// TwinCAT 3 PLC project PLC
// ProgramVersion: 3.1.4023.0
// libraries:
//   Tc2_Standard, * (Beckhoff Automation GmbH)
//   Tc2_System, * (Beckhoff Automation GmbH)
//   Tc3_Module, * (Beckhoff Automation GmbH)
// project tree:
//   / PlcTask.TcTTO
//   POUs/ MAIN.TcPOU
//   DUTs/IO/PdoEntries/ Status_543010BE.TcDUT, Samples_F24E104A.TcDUT, StartTimeNextLatch_02E0C1C8.TcDUT, Status_06143A9F.TcDUT, Status_BA3D1C5D.TcDUT, Status_F2CE6D91.TcDUT, Control_EBEDCF76.TcDUT
//   DUTs/IO/PDOs/ InfoData_6F19DB2B.TcDUT, PAI_Status_Channel_AE4AC104.TcDUT, PAI_Samples_1_Channel_EEA51725.TcDUT, PAI_Timestamp_Channel_6DC4D296.TcDUT, WcState_9091E0EB.TcDUT, InfoData_BEF6B88E.TcDUT, MMS_Device_Inputs_7D6F8734.TcDUT, MMS_Acceleration_Status_11769099.TcDUT, MMS_Acceleration_X_Axis_80E77D6A.TcDUT, MMS_Acceleration_Y_Axis_80E77D6A.TcDUT, MMS_Acceleration_Z_Axis_80E77D6A.TcDUT, MMS_Acceleration_Timestamp_8B9FE1A2.TcDUT, MMS_Voltage_Us_In_Inputs_60D55C72.TcDUT, MMS_Voltage_Up_In_Inputs_60D55C72.TcDUT, MMS_Voltage_Up_Out_Inputs_60D55C72.TcDUT, MMS_Device_Outputs_E6E6F9D1.TcDUT, InfoData_E68C61CD.TcDUT, WcState_0B2B16F9.TcDUT, InfoData_2A97D6CF.TcDUT, Inputs_25A0042B.TcDUT, Outputs_2397A10E.TcDUT
//   DUTs/IO/Boxes/ EK1100_1FC0878B.TcDUT, EK1122_1FC0878B.TcDUT, ELM3002_B416BFEF.TcDUT, ELM3004_9E251EA4.TcDUT, ELM3102_B416BFEF.TcDUT, ELM3104_9E251EA4.TcDUT, ELM3142_B416BFEF.TcDUT, ELM3144_9E251EA4.TcDUT, ELM3146_EA6DB5D7.TcDUT, ELM3148_0838C628.TcDUT, ELM3502_B416BFEF.TcDUT, ELM3504_9E251EA4.TcDUT, ELM3602_B416BFEF.TcDUT, ELM3604_9E251EA4.TcDUT, ELM3702_B416BFEF.TcDUT, ELM3704_9E251EA4.TcDUT, ELM9410_DD553935.TcDUT
//   DUTs/IO/Devices/ SyncUnitTask_2D604ED5.TcDUT, SyncUnitTasks_6FEB8257.TcDUT, SyncUnits_99E584AF.TcDUT
//   DUTs/IO/Topology/ Beckhoff_ELM3xxxEK1122_1A0BF035.TcDUT, Beckhoff_ELM3xxx_31A44528.TcDUT, Beckhoff_ELM31xxEK1122_DD495580.TcDUT, Beckhoff_ELM31xx_96F66E1E.TcDUT, Beckhoff_ELM35xxEK1122_0F7152EB.TcDUT, Beckhoff_ELM35xx_B8844D22.TcDUT, Beckhoff_ELM36xxEK1122_91B39932.TcDUT, Beckhoff_ELM36xx_2C7C6FAB.TcDUT, Beckhoff_ELM37xxEK1122_E40DDF85.TcDUT, Beckhoff_ELM37xx_73C6C048.TcDUT, Beckhoff_ELM3xxx_0030EK1122_95B17030.TcDUT, Beckhoff_ELM3xxx_0030_615BF1E1.TcDUT, Beckhoff_ELM9xxxEK1122_C8584423.TcDUT, Beckhoff_ELM9xxx_3A75798B.TcDUT, EtherCAT_Master_ELMxxxx_56F7A9AD.TcDUT
//   DUTs/IO/Base/ EtcSlaveBase_82538BE2.TcDUT, EtcSlaveBase_82538BE2.TcDUT, EtcSlaveBase_82538BE2.TcDUT, EtcSlaveTerminalBase_947E5A46.TcDUT, EtcSlaveBoxBase_77A0E4A7.TcDUT, EtcSlaveEndTerminalBase_866C7F0C.TcDUT, InputBase_8311D824.TcDUT, OutputBase_10CEE7DE.TcDUT, EtcMasterBase_62654B43.TcDUT
//   GVLs/ GVL_iXlinker.TcGVL

CONFIGURATION PLC
    RESOURCE PLC ON TwinCAT3
        TASK PlcTask(INTERVAL := T#10ms, PRIORITY := 20);
        PROGRAM MAIN WITH PlcTask : MAIN;
    END_RESOURCE
END_CONFIGURATION

// ---- DUTs/IO/PdoEntries/Status_543010BE.TcDUT
{attribute 'GeneratedUsingTerminal: ELM3002-0000-0016'}
{attribute addProperty BoxType "ELM3002-0000-0016"}
{attribute addProperty Id "No_of_SamplesUSINT1ErrorBOOL1UnderrangeBOOL1OverrangeBOOL1DiagBOOL1TxPDO_StateBOOL1Input_cycle_counterBYTE1"}
{attribute addProperty CRC "1412436158"}
{attribute addProperty Size "7"}
TYPE Status_543010BE :
STRUCT
	{attribute addProperty Name "No_of_Samples"}
	No_of_Samples : USINT;
	{attribute addProperty Name "Error"}
	Error : BOOL;
	{attribute addProperty Name "Underrange"}
	Underrange : BOOL;
	{attribute addProperty Name "Overrange"}
	Overrange : BOOL;
	{attribute addProperty Name "Diag"}
	Diag : BOOL;
	{attribute addProperty Name "TxPDO_State"}
	TxPDO_State : BOOL;
	{attribute addProperty Name "Input_cycle_counter"}
	Input_cycle_counter : BYTE;
END_STRUCT
END_TYPE

// ---- DUTs/IO/PdoEntries/Samples_F24E104A.TcDUT
{attribute 'GeneratedUsingTerminal: ELM3002-0000-0016'}
{attribute addProperty BoxType "ELM3002-0000-0016"}
{attribute addProperty Id "ARRAY_0DINT4"}
{attribute addProperty CRC "4065202250"}
{attribute addProperty Size "4"}
TYPE Samples_F24E104A :
STRUCT
	{attribute addProperty Name "ARRAY_0"}
	ARRAY_0 : DINT;
END_STRUCT
END_TYPE

// ---- DUTs/IO/PdoEntries/StartTimeNextLatch_02E0C1C8.TcDUT
{attribute 'GeneratedUsingTerminal: ELM3002-0000-0016'}
{attribute addProperty BoxType "ELM3002-0000-0016"}
{attribute addProperty Id "LowUDINT4HiUDINT4"}
{attribute addProperty CRC "48284104"}
{attribute addProperty Size "8"}
TYPE StartTimeNextLatch_02E0C1C8 :
STRUCT
	{attribute addProperty Name "Low"}
	Low : UDINT;
	{attribute addProperty Name "Hi"}
	Hi : UDINT;
END_STRUCT
END_TYPE

// ---- DUTs/IO/PdoEntries/Status_06143A9F.TcDUT
{attribute 'GeneratedUsingTerminal: ELM9410-0000-0016'}
{attribute addProperty BoxType "ELM9410-0000-0016"}
{attribute addProperty Id "DiagBOOL1ErrorBOOL1Input_cycle_CounterBYTE1TxPDO_StateBOOL1"}
{attribute addProperty CRC "101989023"}
{attribute addProperty Size "4"}
TYPE Status_06143A9F :
STRUCT
	{attribute addProperty Name "Diag"}
	Diag : BOOL;
	{attribute addProperty Name "Error"}
	Error : BOOL;
	{attribute addProperty Name "Input_cycle_Counter"}
	Input_cycle_Counter : BYTE;
	{attribute addProperty Name "TxPDO_State"}
	TxPDO_State : BOOL;
END_STRUCT
END_TYPE

// ---- DUTs/IO/PdoEntries/Status_BA3D1C5D.TcDUT
{attribute 'GeneratedUsingTerminal: ELM9410-0000-0016'}
{attribute addProperty BoxType "ELM9410-0000-0016"}
{attribute addProperty Id "ErrorBOOL1UnderrangeBOOL1OverrangeBOOL1DiagBOOL1Sensor_OvrBOOL1OverrunBOOL1TxPDO_StateBOOL1"}
{attribute addProperty CRC "3124567133"}
{attribute addProperty Size "7"}
TYPE Status_BA3D1C5D :
STRUCT
	{attribute addProperty Name "Error"}
	Error : BOOL;
	{attribute addProperty Name "Underrange"}
	Underrange : BOOL;
	{attribute addProperty Name "Overrange"}
	Overrange : BOOL;
	{attribute addProperty Name "Diag"}
	Diag : BOOL;
	{attribute addProperty Name "Sensor_Ovr"}
	Sensor_Ovr : BOOL;
	{attribute addProperty Name "Overrun"}
	Overrun : BOOL;
	{attribute addProperty Name "TxPDO_State"}
	TxPDO_State : BOOL;
END_STRUCT
END_TYPE

// ---- DUTs/IO/PdoEntries/Status_F2CE6D91.TcDUT
{attribute 'GeneratedUsingTerminal: ELM9410-0000-0016'}
{attribute addProperty BoxType "ELM9410-0000-0016"}
{attribute addProperty Id "UnderrangeBOOL1OverrangeBOOL1Limit_1BYTE1Limit_2BYTE1ErrorBOOL1TxPDO_StateBOOL1TxPDO_ToggleBOOL1"}
{attribute addProperty CRC "4073614737"}
{attribute addProperty Size "7"}
TYPE Status_F2CE6D91 :
STRUCT
	{attribute addProperty Name "Underrange"}
	Underrange : BOOL;
	{attribute addProperty Name "Overrange"}
	Overrange : BOOL;
	{attribute addProperty Name "Limit_1"}
	Limit_1 : BYTE;
	{attribute addProperty Name "Limit_2"}
	Limit_2 : BYTE;
	{attribute addProperty Name "Error"}
	Error : BOOL;
	{attribute addProperty Name "TxPDO_State"}
	TxPDO_State : BOOL;
	{attribute addProperty Name "TxPDO_Toggle"}
	TxPDO_Toggle : BOOL;
END_STRUCT
END_TYPE

// ---- DUTs/IO/PdoEntries/Control_EBEDCF76.TcDUT
{attribute 'GeneratedUsingTerminal: ELM9410-0000-0016'}
{attribute addProperty BoxType "ELM9410-0000-0016"}
{attribute addProperty Id "Up_Out_OFFBOOL1"}
{attribute addProperty CRC "3958230902"}
{attribute addProperty Size "1"}
TYPE Control_EBEDCF76 :
STRUCT
	{attribute addProperty Name "Up_Out_OFF"}
	Up_Out_OFF : BOOL;
END_STRUCT
END_TYPE

// ---- DUTs/IO/PDOs/InfoData_6F19DB2B.TcDUT
{attribute 'GeneratedUsingTerminal: EK1100-0000-0018'}
{attribute addProperty BoxType "EK1100-0000-0018"}
{attribute addProperty Id "StateAT %I*UINT2"}
{attribute addProperty CRC "1863965483"}
{attribute addProperty Size "2"}
TYPE InfoData_6F19DB2B :
STRUCT
	{attribute addProperty Name "State"}
	State AT %I* : UINT;
END_STRUCT
END_TYPE

// ---- DUTs/IO/PDOs/PAI_Status_Channel_AE4AC104.TcDUT
{attribute 'GeneratedUsingTerminal: ELM3002-0000-0016'}
{attribute addProperty BoxType "ELM3002-0000-0016"}
{attribute addProperty Id "StatusAT %I*Status_543010BE7"}
{attribute addProperty CRC "2924134660"}
{attribute addProperty Size "7"}
TYPE PAI_Status_Channel_AE4AC104 EXTENDS InputBase_8311D824 :
STRUCT
	{attribute addProperty Name "Status"}
	Status AT %I* : Status_543010BE;
END_STRUCT
END_TYPE

// ---- DUTs/IO/PDOs/PAI_Samples_1_Channel_EEA51725.TcDUT
{attribute 'GeneratedUsingTerminal: ELM3002-0000-0016'}
{attribute addProperty BoxType "ELM3002-0000-0016"}
{attribute addProperty Id "SamplesAT %I*Samples_F24E104A4"}
{attribute addProperty CRC "4003796773"}
{attribute addProperty Size "4"}
TYPE PAI_Samples_1_Channel_EEA51725 EXTENDS InputBase_8311D824 :
STRUCT
	{attribute addProperty Name "Samples"}
	Samples AT %I* : Samples_F24E104A;
END_STRUCT
END_TYPE

// ---- DUTs/IO/PDOs/PAI_Timestamp_Channel_6DC4D296.TcDUT
{attribute 'GeneratedUsingTerminal: ELM3002-0000-0016'}
{attribute addProperty BoxType "ELM3002-0000-0016"}
{attribute addProperty Id "StartTimeNextLatchAT %I*StartTimeNextLatch_02E0C1C88"}
{attribute addProperty CRC "1841615510"}
{attribute addProperty Size "8"}
TYPE PAI_Timestamp_Channel_6DC4D296 EXTENDS InputBase_8311D824 :
STRUCT
	{attribute addProperty Name "StartTimeNextLatch"}
	StartTimeNextLatch AT %I* : StartTimeNextLatch_02E0C1C8;
END_STRUCT
END_TYPE

// ---- DUTs/IO/PDOs/WcState_9091E0EB.TcDUT
{attribute 'GeneratedUsingTerminal: ELM3002-0000-0016'}
{attribute addProperty BoxType "ELM3002-0000-0016"}
{attribute addProperty Id "WcStateAT %I*BOOL1InputToggleAT %I*BOOL1"}
{attribute addProperty CRC "2425479403"}
{attribute addProperty Size "2"}
TYPE WcState_9091E0EB :
STRUCT
	{attribute addProperty Name "WcState"}
	WcState AT %I* : BOOL;
	{attribute addProperty Name "InputToggle"}
	InputToggle AT %I* : BOOL;
END_STRUCT
END_TYPE

// ---- DUTs/IO/PDOs/InfoData_BEF6B88E.TcDUT
{attribute 'GeneratedUsingTerminal: ELM3002-0000-0016'}
{attribute addProperty BoxType "ELM3002-0000-0016"}
{attribute addProperty Id "AdsAddrAT %I*AMSADDR8DcOutputShiftAT %I*DINT4DcInputShiftAT %I*DINT4StateAT %I*UINT2"}
{attribute addProperty CRC "3203840142"}
{attribute addProperty Size "18"}
TYPE InfoData_BEF6B88E EXTENDS InputBase_8311D824 :
STRUCT
	{attribute addProperty Name "AdsAddr"}
	AdsAddr AT %I* : AMSADDR;
	{attribute addProperty Name "DcOutputShift"}
	DcOutputShift AT %I* : DINT;
	{attribute addProperty Name "DcInputShift"}
	DcInputShift AT %I* : DINT;
	{attribute addProperty Name "State"}
	State AT %I* : UINT;
END_STRUCT
END_TYPE

// ---- DUTs/IO/PDOs/MMS_Device_Inputs_7D6F8734.TcDUT
{attribute 'GeneratedUsingTerminal: ELM9410-0000-0016'}
{attribute addProperty BoxType "ELM9410-0000-0016"}
{attribute addProperty Id "StatusAT %I*Status_06143A9F4"}
{attribute addProperty CRC "2104461108"}
{attribute addProperty Size "4"}
TYPE MMS_Device_Inputs_7D6F8734 EXTENDS InputBase_8311D824 :
STRUCT
	{attribute addProperty Name "Status"}
	Status AT %I* : Status_06143A9F;
END_STRUCT
END_TYPE

// ---- DUTs/IO/PDOs/MMS_Acceleration_Status_11769099.TcDUT
{attribute 'GeneratedUsingTerminal: ELM9410-0000-0016'}
{attribute addProperty BoxType "ELM9410-0000-0016"}
{attribute addProperty Id "StatusAT %I*Status_BA3D1C5D7Number_of_samplesAT %I*UINT2"}
{attribute addProperty CRC "292982937"}
{attribute addProperty Size "9"}
TYPE MMS_Acceleration_Status_11769099 EXTENDS InputBase_8311D824 :
STRUCT
	{attribute addProperty Name "Status"}
	Status AT %I* : Status_BA3D1C5D;
	{attribute addProperty Name "Number_of_samples"}
	Number_of_samples AT %I* : UINT;
END_STRUCT
END_TYPE

// ---- DUTs/IO/PDOs/MMS_Acceleration_X_Axis_80E77D6A.TcDUT
{attribute 'GeneratedUsingTerminal: ELM9410-0000-0016'}
{attribute addProperty BoxType "ELM9410-0000-0016"}
{attribute addProperty Id "ValueAT %I*INT2"}
{attribute addProperty CRC "2162654570"}
{attribute addProperty Size "2"}
TYPE MMS_Acceleration_X_Axis_80E77D6A EXTENDS InputBase_8311D824 :
STRUCT
	{attribute addProperty Name "Value"}
	Value AT %I* : INT;
END_STRUCT
END_TYPE

// ---- DUTs/IO/PDOs/MMS_Acceleration_Y_Axis_80E77D6A.TcDUT
{attribute 'GeneratedUsingTerminal: ELM9410-0000-0016'}
{attribute addProperty BoxType "ELM9410-0000-0016"}
{attribute addProperty Id "ValueAT %I*INT2"}
{attribute addProperty CRC "2162654570"}
{attribute addProperty Size "2"}
TYPE MMS_Acceleration_Y_Axis_80E77D6A EXTENDS InputBase_8311D824 :
STRUCT
	{attribute addProperty Name "Value"}
	Value AT %I* : INT;
END_STRUCT
END_TYPE

// ---- DUTs/IO/PDOs/MMS_Acceleration_Z_Axis_80E77D6A.TcDUT
{attribute 'GeneratedUsingTerminal: ELM9410-0000-0016'}
{attribute addProperty BoxType "ELM9410-0000-0016"}
{attribute addProperty Id "ValueAT %I*INT2"}
{attribute addProperty CRC "2162654570"}
{attribute addProperty Size "2"}
TYPE MMS_Acceleration_Z_Axis_80E77D6A EXTENDS InputBase_8311D824 :
STRUCT
	{attribute addProperty Name "Value"}
	Value AT %I* : INT;
END_STRUCT
END_TYPE

// ---- DUTs/IO/PDOs/MMS_Acceleration_Timestamp_8B9FE1A2.TcDUT
{attribute 'GeneratedUsingTerminal: ELM9410-0000-0016'}
{attribute addProperty BoxType "ELM9410-0000-0016"}
{attribute addProperty Id "TimestampAT %I*ULINT8"}
{attribute addProperty CRC "2342511010"}
{attribute addProperty Size "8"}
TYPE MMS_Acceleration_Timestamp_8B9FE1A2 EXTENDS InputBase_8311D824 :
STRUCT
	{attribute addProperty Name "Timestamp"}
	Timestamp AT %I* : ULINT;
END_STRUCT
END_TYPE

// ---- DUTs/IO/PDOs/MMS_Voltage_Us_In_Inputs_60D55C72.TcDUT
{attribute 'GeneratedUsingTerminal: ELM9410-0000-0016'}
{attribute addProperty BoxType "ELM9410-0000-0016"}
{attribute addProperty Id "StatusAT %I*Status_F2CE6D917ValueAT %I*REAL4"}
{attribute addProperty CRC "1624595570"}
{attribute addProperty Size "11"}
TYPE MMS_Voltage_Us_In_Inputs_60D55C72 EXTENDS InputBase_8311D824 :
STRUCT
	{attribute addProperty Name "Status"}
	Status AT %I* : Status_F2CE6D91;
	{attribute addProperty Name "Value"}
	Value AT %I* : REAL;
END_STRUCT
END_TYPE

// ---- DUTs/IO/PDOs/MMS_Voltage_Up_In_Inputs_60D55C72.TcDUT
{attribute 'GeneratedUsingTerminal: ELM9410-0000-0016'}
{attribute addProperty BoxType "ELM9410-0000-0016"}
{attribute addProperty Id "StatusAT %I*Status_F2CE6D917ValueAT %I*REAL4"}
{attribute addProperty CRC "1624595570"}
{attribute addProperty Size "11"}
TYPE MMS_Voltage_Up_In_Inputs_60D55C72 EXTENDS InputBase_8311D824 :
STRUCT
	{attribute addProperty Name "Status"}
	Status AT %I* : Status_F2CE6D91;
	{attribute addProperty Name "Value"}
	Value AT %I* : REAL;
END_STRUCT
END_TYPE

// ---- DUTs/IO/PDOs/MMS_Voltage_Up_Out_Inputs_60D55C72.TcDUT
{attribute 'GeneratedUsingTerminal: ELM9410-0000-0016'}
{attribute addProperty BoxType "ELM9410-0000-0016"}
{attribute addProperty Id "StatusAT %I*Status_F2CE6D917ValueAT %I*REAL4"}
{attribute addProperty CRC "1624595570"}
{attribute addProperty Size "11"}
TYPE MMS_Voltage_Up_Out_Inputs_60D55C72 EXTENDS InputBase_8311D824 :
STRUCT
	{attribute addProperty Name "Status"}
	Status AT %I* : Status_F2CE6D91;
	{attribute addProperty Name "Value"}
	Value AT %I* : REAL;
END_STRUCT
END_TYPE

// ---- DUTs/IO/PDOs/MMS_Device_Outputs_E6E6F9D1.TcDUT
{attribute 'GeneratedUsingTerminal: ELM9410-0000-0016'}
{attribute addProperty BoxType "ELM9410-0000-0016"}
{attribute addProperty Id "ControlAT %Q*Control_EBEDCF761"}
{attribute addProperty CRC "3873896913"}
{attribute addProperty Size "1"}
TYPE MMS_Device_Outputs_E6E6F9D1 EXTENDS OutputBase_10CEE7DE :
STRUCT
	{attribute addProperty Name "Control"}
	Control AT %Q* : Control_EBEDCF76;
END_STRUCT
END_TYPE

// ---- DUTs/IO/PDOs/InfoData_E68C61CD.TcDUT
{attribute 'GeneratedUsingTerminal: IODEVICETYPE_ETHERCATPROT'}
{attribute addProperty BoxType "IODEVICETYPE_ETHERCATPROT"}
{attribute addProperty Id "ChangeCountAT %I*UINT2DevIdAT %I*UINT2AmsNetIdAT %I*AMSNETID6CfgSlaveCountAT %I*UINT2DcToTcTimeOffsetAT %I*LINT8DcToExtTimeOffsetAT %I*LINT8"}
{attribute addProperty CRC "3867959757"}
{attribute addProperty Size "28"}
TYPE InfoData_E68C61CD EXTENDS InputBase_8311D824 :
STRUCT
	{attribute addProperty Name "ChangeCount"}
	ChangeCount AT %I* : UINT;
	{attribute addProperty Name "DevId"}
	DevId AT %I* : UINT;
	{attribute addProperty Name "AmsNetId"}
	AmsNetId AT %I* : AMSNETID;
	{attribute addProperty Name "CfgSlaveCount"}
	CfgSlaveCount AT %I* : UINT;
	{attribute addProperty Name "DcToTcTimeOffset"}
	DcToTcTimeOffset AT %I* : LINT;
	{attribute addProperty Name "DcToExtTimeOffset"}
	DcToExtTimeOffset AT %I* : LINT;
END_STRUCT
END_TYPE

// ---- DUTs/IO/PDOs/WcState_0B2B16F9.TcDUT
{attribute 'GeneratedUsingTerminal: IODEVICETYPE_ETHERCATPROT'}
{attribute addProperty BoxType "IODEVICETYPE_ETHERCATPROT"}
{attribute addProperty Id "WcStateAT %I*BOOL1"}
{attribute addProperty CRC "187373305"}
{attribute addProperty Size "1"}
TYPE WcState_0B2B16F9 :
STRUCT
	{attribute addProperty Name "WcState"}
	WcState AT %I* : BOOL;
END_STRUCT
END_TYPE

// ---- DUTs/IO/PDOs/InfoData_2A97D6CF.TcDUT
{attribute 'GeneratedUsingTerminal: IODEVICETYPE_ETHERCATPROT'}
{attribute addProperty BoxType "IODEVICETYPE_ETHERCATPROT"}
{attribute addProperty Id "ObjectIdAT %I*OTCID4StateAT %I*UINT2SlaveCountAT %I*UINT2"}
{attribute addProperty CRC "714593999"}
{attribute addProperty Size "8"}
TYPE InfoData_2A97D6CF EXTENDS InputBase_8311D824 :
STRUCT
	{attribute addProperty Name "ObjectId"}
	ObjectId AT %I* : OTCID;
	{attribute addProperty Name "State"}
	State AT %I* : UINT;
	{attribute addProperty Name "SlaveCount"}
	SlaveCount AT %I* : UINT;
END_STRUCT
END_TYPE

// ---- DUTs/IO/PDOs/Inputs_25A0042B.TcDUT
{attribute 'GeneratedUsingTerminal: IODEVICETYPE_ETHERCATPROT'}
{attribute addProperty BoxType "IODEVICETYPE_ETHERCATPROT"}
{attribute addProperty Id "SlaveCountAT %I*UINT2DevStateAT %I*UINT2Frm0StateAT %I*UINT2Frm0WcStateAT %I*UINT2Frm0InputToggleAT %I*UINT2Frm1StateAT %I*UINT2Frm1WcStateAT %I*UINT2Frm1InputToggleAT %I*UINT2Frm2StateAT %I*UINT2Frm2WcStateAT %I*UINT2Frm2InputToggleAT %I*UINT2Frm3StateAT %I*UINT2Frm3WcStateAT %I*UINT2Frm3InputToggleAT %I*UINT2Frm4StateAT %I*UINT2Frm4WcStateAT %I*UINT2Frm4InputToggleAT %I*UINT2Frm5StateAT %I*UINT2Frm5WcStateAT %I*UINT2Frm5InputToggleAT %I*UINT2Frm6StateAT %I*UINT2Frm6WcStateAT %I*UINT2Frm6InputToggleAT %I*UINT2Frm7StateAT %I*UINT2Frm7WcStateAT %I*UINT2Frm7InputToggleAT %I*UINT2Frm8StateAT %I*UINT2Frm8WcStateAT %I*UINT2Frm8InputToggleAT %I*UINT2Frm9StateAT %I*UINT2Frm9WcStateAT %I*UINT2Frm9InputToggleAT %I*UINT2Frm10StateAT %I*UINT2Frm10WcStateAT %I*UINT2Frm10InputToggleAT %I*UINT2Frm11StateAT %I*UINT2Frm11WcStateAT %I*UINT2Frm11InputToggleAT %I*UINT2Frm12StateAT %I*UINT2Frm12WcStateAT %I*UINT2Frm12InputToggleAT %I*UINT2Frm13StateAT %I*UINT2Frm13WcStateAT %I*UINT2Frm13InputToggleAT %I*UINT2Frm14StateAT %I*UINT2Frm14WcStateAT %I*UINT2Frm14InputToggleAT %I*UINT2Frm15StateAT %I*UINT2Frm15WcStateAT %I*UINT2Frm15InputToggleAT %I*UINT2Frm16StateAT %I*UINT2Frm16WcStateAT %I*UINT2Frm16InputToggleAT %I*UINT2Frm17StateAT %I*UINT2Frm17WcStateAT %I*UINT2Frm17InputToggleAT %I*UINT2Frm18StateAT %I*UINT2Frm18WcStateAT %I*UINT2Frm18InputToggleAT %I*UINT2Frm19StateAT %I*UINT2Frm19WcStateAT %I*UINT2Frm19InputToggleAT %I*UINT2Frm20StateAT %I*UINT2Frm20WcStateAT %I*UINT2Frm20InputToggleAT %I*UINT2Frm21StateAT %I*UINT2Frm21WcStateAT %I*UINT2Frm21InputToggleAT %I*UINT2Frm22StateAT %I*UINT2Frm22WcStateAT %I*UINT2Frm22InputToggleAT %I*UINT2Frm23StateAT %I*UINT2Frm23WcStateAT %I*UINT2Frm23InputToggleAT %I*UINT2Frm24StateAT %I*UINT2Frm24WcStateAT %I*UINT2Frm24InputToggleAT %I*UINT2Frm25StateAT %I*UINT2Frm25WcStateAT %I*UINT2Frm25InputToggleAT %I*UINT2"}
{attribute addProperty CRC "631243819"}
{attribute addProperty Size "160"}
TYPE Inputs_25A0042B EXTENDS InputBase_8311D824 :
STRUCT
	{attribute addProperty Name "SlaveCount"}
	SlaveCount AT %I* : UINT;
	{attribute addProperty Name "DevState"}
	DevState AT %I* : UINT;
	{attribute addProperty Name "Frm0State"}
	Frm0State AT %I* : UINT;
	{attribute addProperty Name "Frm0WcState"}
	Frm0WcState AT %I* : UINT;
	{attribute addProperty Name "Frm0InputToggle"}
	Frm0InputToggle AT %I* : UINT;
	{attribute addProperty Name "Frm1State"}
	Frm1State AT %I* : UINT;
	{attribute addProperty Name "Frm1WcState"}
	Frm1WcState AT %I* : UINT;
	{attribute addProperty Name "Frm1InputToggle"}
	Frm1InputToggle AT %I* : UINT;
	{attribute addProperty Name "Frm2State"}
	Frm2State AT %I* : UINT;
	{attribute addProperty Name "Frm2WcState"}
	Frm2WcState AT %I* : UINT;
	{attribute addProperty Name "Frm2InputToggle"}
	Frm2InputToggle AT %I* : UINT;
	{attribute addProperty Name "Frm3State"}
	Frm3State AT %I* : UINT;
	{attribute addProperty Name "Frm3WcState"}
	Frm3WcState AT %I* : UINT;
	{attribute addProperty Name "Frm3InputToggle"}
	Frm3InputToggle AT %I* : UINT;
	{attribute addProperty Name "Frm4State"}
	Frm4State AT %I* : UINT;
	{attribute addProperty Name "Frm4WcState"}
	Frm4WcState AT %I* : UINT;
	{attribute addProperty Name "Frm4InputToggle"}
	Frm4InputToggle AT %I* : UINT;
	{attribute addProperty Name "Frm5State"}
	Frm5State AT %I* : UINT;
	{attribute addProperty Name "Frm5WcState"}
	Frm5WcState AT %I* : UINT;
	{attribute addProperty Name "Frm5InputToggle"}
	Frm5InputToggle AT %I* : UINT;
	{attribute addProperty Name "Frm6State"}
	Frm6State AT %I* : UINT;
	{attribute addProperty Name "Frm6WcState"}
	Frm6WcState AT %I* : UINT;
	{attribute addProperty Name "Frm6InputToggle"}
	Frm6InputToggle AT %I* : UINT;
	{attribute addProperty Name "Frm7State"}
	Frm7State AT %I* : UINT;
	{attribute addProperty Name "Frm7WcState"}
	Frm7WcState AT %I* : UINT;
	{attribute addProperty Name "Frm7InputToggle"}
	Frm7InputToggle AT %I* : UINT;
	{attribute addProperty Name "Frm8State"}
	Frm8State AT %I* : UINT;
	{attribute addProperty Name "Frm8WcState"}
	Frm8WcState AT %I* : UINT;
	{attribute addProperty Name "Frm8InputToggle"}
	Frm8InputToggle AT %I* : UINT;
	{attribute addProperty Name "Frm9State"}
	Frm9State AT %I* : UINT;
	{attribute addProperty Name "Frm9WcState"}
	Frm9WcState AT %I* : UINT;
	{attribute addProperty Name "Frm9InputToggle"}
	Frm9InputToggle AT %I* : UINT;
	{attribute addProperty Name "Frm10State"}
	Frm10State AT %I* : UINT;
	{attribute addProperty Name "Frm10WcState"}
	Frm10WcState AT %I* : UINT;
	{attribute addProperty Name "Frm10InputToggle"}
	Frm10InputToggle AT %I* : UINT;
	{attribute addProperty Name "Frm11State"}
	Frm11State AT %I* : UINT;
	{attribute addProperty Name "Frm11WcState"}
	Frm11WcState AT %I* : UINT;
	{attribute addProperty Name "Frm11InputToggle"}
	Frm11InputToggle AT %I* : UINT;
	{attribute addProperty Name "Frm12State"}
	Frm12State AT %I* : UINT;
	{attribute addProperty Name "Frm12WcState"}
	Frm12WcState AT %I* : UINT;
	{attribute addProperty Name "Frm12InputToggle"}
	Frm12InputToggle AT %I* : UINT;
	{attribute addProperty Name "Frm13State"}
	Frm13State AT %I* : UINT;
	{attribute addProperty Name "Frm13WcState"}
	Frm13WcState AT %I* : UINT;
	{attribute addProperty Name "Frm13InputToggle"}
	Frm13InputToggle AT %I* : UINT;
	{attribute addProperty Name "Frm14State"}
	Frm14State AT %I* : UINT;
	{attribute addProperty Name "Frm14WcState"}
	Frm14WcState AT %I* : UINT;
	{attribute addProperty Name "Frm14InputToggle"}
	Frm14InputToggle AT %I* : UINT;
	{attribute addProperty Name "Frm15State"}
	Frm15State AT %I* : UINT;
	{attribute addProperty Name "Frm15WcState"}
	Frm15WcState AT %I* : UINT;
	{attribute addProperty Name "Frm15InputToggle"}
	Frm15InputToggle AT %I* : UINT;
	{attribute addProperty Name "Frm16State"}
	Frm16State AT %I* : UINT;
	{attribute addProperty Name "Frm16WcState"}
	Frm16WcState AT %I* : UINT;
	{attribute addProperty Name "Frm16InputToggle"}
	Frm16InputToggle AT %I* : UINT;
	{attribute addProperty Name "Frm17State"}
	Frm17State AT %I* : UINT;
	{attribute addProperty Name "Frm17WcState"}
	Frm17WcState AT %I* : UINT;
	{attribute addProperty Name "Frm17InputToggle"}
	Frm17InputToggle AT %I* : UINT;
	{attribute addProperty Name "Frm18State"}
	Frm18State AT %I* : UINT;
	{attribute addProperty Name "Frm18WcState"}
	Frm18WcState AT %I* : UINT;
	{attribute addProperty Name "Frm18InputToggle"}
	Frm18InputToggle AT %I* : UINT;
	{attribute addProperty Name "Frm19State"}
	Frm19State AT %I* : UINT;
	{attribute addProperty Name "Frm19WcState"}
	Frm19WcState AT %I* : UINT;
	{attribute addProperty Name "Frm19InputToggle"}
	Frm19InputToggle AT %I* : UINT;
	{attribute addProperty Name "Frm20State"}
	Frm20State AT %I* : UINT;
	{attribute addProperty Name "Frm20WcState"}
	Frm20WcState AT %I* : UINT;
	{attribute addProperty Name "Frm20InputToggle"}
	Frm20InputToggle AT %I* : UINT;
	{attribute addProperty Name "Frm21State"}
	Frm21State AT %I* : UINT;
	{attribute addProperty Name "Frm21WcState"}
	Frm21WcState AT %I* : UINT;
	{attribute addProperty Name "Frm21InputToggle"}
	Frm21InputToggle AT %I* : UINT;
	{attribute addProperty Name "Frm22State"}
	Frm22State AT %I* : UINT;
	{attribute addProperty Name "Frm22WcState"}
	Frm22WcState AT %I* : UINT;
	{attribute addProperty Name "Frm22InputToggle"}
	Frm22InputToggle AT %I* : UINT;
	{attribute addProperty Name "Frm23State"}
	Frm23State AT %I* : UINT;
	{attribute addProperty Name "Frm23WcState"}
	Frm23WcState AT %I* : UINT;
	{attribute addProperty Name "Frm23InputToggle"}
	Frm23InputToggle AT %I* : UINT;
	{attribute addProperty Name "Frm24State"}
	Frm24State AT %I* : UINT;
	{attribute addProperty Name "Frm24WcState"}
	Frm24WcState AT %I* : UINT;
	{attribute addProperty Name "Frm24InputToggle"}
	Frm24InputToggle AT %I* : UINT;
	{attribute addProperty Name "Frm25State"}
	Frm25State AT %I* : UINT;
	{attribute addProperty Name "Frm25WcState"}
	Frm25WcState AT %I* : UINT;
	{attribute addProperty Name "Frm25InputToggle"}
	Frm25InputToggle AT %I* : UINT;
END_STRUCT
END_TYPE

// ---- DUTs/IO/PDOs/Outputs_2397A10E.TcDUT
{attribute 'GeneratedUsingTerminal: IODEVICETYPE_ETHERCATPROT'}
{attribute addProperty BoxType "IODEVICETYPE_ETHERCATPROT"}
{attribute addProperty Id "DevCtrlAT %Q*UINT2Frm0CtrlAT %Q*UINT2Frm0WcCtrlAT %Q*UINT2Frm1CtrlAT %Q*UINT2Frm1WcCtrlAT %Q*UINT2Frm2CtrlAT %Q*UINT2Frm2WcCtrlAT %Q*UINT2Frm3CtrlAT %Q*UINT2Frm3WcCtrlAT %Q*UINT2Frm4CtrlAT %Q*UINT2Frm4WcCtrlAT %Q*UINT2Frm5CtrlAT %Q*UINT2Frm5WcCtrlAT %Q*UINT2Frm6CtrlAT %Q*UINT2Frm6WcCtrlAT %Q*UINT2Frm7CtrlAT %Q*UINT2Frm7WcCtrlAT %Q*UINT2Frm8CtrlAT %Q*UINT2Frm8WcCtrlAT %Q*UINT2Frm9CtrlAT %Q*UINT2Frm9WcCtrlAT %Q*UINT2Frm10CtrlAT %Q*UINT2Frm10WcCtrlAT %Q*UINT2Frm11CtrlAT %Q*UINT2Frm11WcCtrlAT %Q*UINT2Frm12CtrlAT %Q*UINT2Frm12WcCtrlAT %Q*UINT2Frm13CtrlAT %Q*UINT2Frm13WcCtrlAT %Q*UINT2Frm14CtrlAT %Q*UINT2Frm14WcCtrlAT %Q*UINT2Frm15CtrlAT %Q*UINT2Frm15WcCtrlAT %Q*UINT2Frm16CtrlAT %Q*UINT2Frm16WcCtrlAT %Q*UINT2Frm17CtrlAT %Q*UINT2Frm17WcCtrlAT %Q*UINT2Frm18CtrlAT %Q*UINT2Frm18WcCtrlAT %Q*UINT2Frm19CtrlAT %Q*UINT2Frm19WcCtrlAT %Q*UINT2Frm20CtrlAT %Q*UINT2Frm20WcCtrlAT %Q*UINT2Frm21CtrlAT %Q*UINT2Frm21WcCtrlAT %Q*UINT2Frm22CtrlAT %Q*UINT2Frm22WcCtrlAT %Q*UINT2Frm23CtrlAT %Q*UINT2Frm23WcCtrlAT %Q*UINT2Frm24CtrlAT %Q*UINT2Frm24WcCtrlAT %Q*UINT2Frm25CtrlAT %Q*UINT2Frm25WcCtrlAT %Q*UINT2"}
{attribute addProperty CRC "597139726"}
{attribute addProperty Size "106"}
TYPE Outputs_2397A10E EXTENDS OutputBase_10CEE7DE :
STRUCT
	{attribute addProperty Name "DevCtrl"}
	DevCtrl AT %Q* : UINT;
	{attribute addProperty Name "Frm0Ctrl"}
	Frm0Ctrl AT %Q* : UINT;
	{attribute addProperty Name "Frm0WcCtrl"}
	Frm0WcCtrl AT %Q* : UINT;
	{attribute addProperty Name "Frm1Ctrl"}
	Frm1Ctrl AT %Q* : UINT;
	{attribute addProperty Name "Frm1WcCtrl"}
	Frm1WcCtrl AT %Q* : UINT;
	{attribute addProperty Name "Frm2Ctrl"}
	Frm2Ctrl AT %Q* : UINT;
	{attribute addProperty Name "Frm2WcCtrl"}
	Frm2WcCtrl AT %Q* : UINT;
	{attribute addProperty Name "Frm3Ctrl"}
	Frm3Ctrl AT %Q* : UINT;
	{attribute addProperty Name "Frm3WcCtrl"}
	Frm3WcCtrl AT %Q* : UINT;
	{attribute addProperty Name "Frm4Ctrl"}
	Frm4Ctrl AT %Q* : UINT;
	{attribute addProperty Name "Frm4WcCtrl"}
	Frm4WcCtrl AT %Q* : UINT;
	{attribute addProperty Name "Frm5Ctrl"}
	Frm5Ctrl AT %Q* : UINT;
	{attribute addProperty Name "Frm5WcCtrl"}
	Frm5WcCtrl AT %Q* : UINT;
	{attribute addProperty Name "Frm6Ctrl"}
	Frm6Ctrl AT %Q* : UINT;
	{attribute addProperty Name "Frm6WcCtrl"}
	Frm6WcCtrl AT %Q* : UINT;
	{attribute addProperty Name "Frm7Ctrl"}
	Frm7Ctrl AT %Q* : UINT;
	{attribute addProperty Name "Frm7WcCtrl"}
	Frm7WcCtrl AT %Q* : UINT;
	{attribute addProperty Name "Frm8Ctrl"}
	Frm8Ctrl AT %Q* : UINT;
	{attribute addProperty Name "Frm8WcCtrl"}
	Frm8WcCtrl AT %Q* : UINT;
	{attribute addProperty Name "Frm9Ctrl"}
	Frm9Ctrl AT %Q* : UINT;
	{attribute addProperty Name "Frm9WcCtrl"}
	Frm9WcCtrl AT %Q* : UINT;
	{attribute addProperty Name "Frm10Ctrl"}
	Frm10Ctrl AT %Q* : UINT;
	{attribute addProperty Name "Frm10WcCtrl"}
	Frm10WcCtrl AT %Q* : UINT;
	{attribute addProperty Name "Frm11Ctrl"}
	Frm11Ctrl AT %Q* : UINT;
	{attribute addProperty Name "Frm11WcCtrl"}
	Frm11WcCtrl AT %Q* : UINT;
	{attribute addProperty Name "Frm12Ctrl"}
	Frm12Ctrl AT %Q* : UINT;
	{attribute addProperty Name "Frm12WcCtrl"}
	Frm12WcCtrl AT %Q* : UINT;
	{attribute addProperty Name "Frm13Ctrl"}
	Frm13Ctrl AT %Q* : UINT;
	{attribute addProperty Name "Frm13WcCtrl"}
	Frm13WcCtrl AT %Q* : UINT;
	{attribute addProperty Name "Frm14Ctrl"}
	Frm14Ctrl AT %Q* : UINT;
	{attribute addProperty Name "Frm14WcCtrl"}
	Frm14WcCtrl AT %Q* : UINT;
	{attribute addProperty Name "Frm15Ctrl"}
	Frm15Ctrl AT %Q* : UINT;
	{attribute addProperty Name "Frm15WcCtrl"}
	Frm15WcCtrl AT %Q* : UINT;
	{attribute addProperty Name "Frm16Ctrl"}
	Frm16Ctrl AT %Q* : UINT;
	{attribute addProperty Name "Frm16WcCtrl"}
	Frm16WcCtrl AT %Q* : UINT;
	{attribute addProperty Name "Frm17Ctrl"}
	Frm17Ctrl AT %Q* : UINT;
	{attribute addProperty Name "Frm17WcCtrl"}
	Frm17WcCtrl AT %Q* : UINT;
	{attribute addProperty Name "Frm18Ctrl"}
	Frm18Ctrl AT %Q* : UINT;
	{attribute addProperty Name "Frm18WcCtrl"}
	Frm18WcCtrl AT %Q* : UINT;
	{attribute addProperty Name "Frm19Ctrl"}
	Frm19Ctrl AT %Q* : UINT;
	{attribute addProperty Name "Frm19WcCtrl"}
	Frm19WcCtrl AT %Q* : UINT;
	{attribute addProperty Name "Frm20Ctrl"}
	Frm20Ctrl AT %Q* : UINT;
	{attribute addProperty Name "Frm20WcCtrl"}
	Frm20WcCtrl AT %Q* : UINT;
	{attribute addProperty Name "Frm21Ctrl"}
	Frm21Ctrl AT %Q* : UINT;
	{attribute addProperty Name "Frm21WcCtrl"}
	Frm21WcCtrl AT %Q* : UINT;
	{attribute addProperty Name "Frm22Ctrl"}
	Frm22Ctrl AT %Q* : UINT;
	{attribute addProperty Name "Frm22WcCtrl"}
	Frm22WcCtrl AT %Q* : UINT;
	{attribute addProperty Name "Frm23Ctrl"}
	Frm23Ctrl AT %Q* : UINT;
	{attribute addProperty Name "Frm23WcCtrl"}
	Frm23WcCtrl AT %Q* : UINT;
	{attribute addProperty Name "Frm24Ctrl"}
	Frm24Ctrl AT %Q* : UINT;
	{attribute addProperty Name "Frm24WcCtrl"}
	Frm24WcCtrl AT %Q* : UINT;
	{attribute addProperty Name "Frm25Ctrl"}
	Frm25Ctrl AT %Q* : UINT;
	{attribute addProperty Name "Frm25WcCtrl"}
	Frm25WcCtrl AT %Q* : UINT;
END_STRUCT
END_TYPE

// ---- DUTs/IO/Boxes/EK1100_1FC0878B.TcDUT
{attribute 'GeneratedUsingTerminal: EK1100-0000-0018'}
{attribute addProperty BoxType "EK1100-0000-0018"}
{attribute addProperty Description "EK1100 EtherCAT Coupler (2A E-Bus)"}
{attribute addProperty Physics "YKY"}
{attribute addProperty Id "InfoDataAT %I*InfoData_6F19DB2B2"}
{attribute addProperty CRC "532711307"}
{attribute addProperty Size "2"}
TYPE EK1100_1FC0878B EXTENDS EtcSlaveBoxBase_77A0E4A7 :
STRUCT
	{attribute addProperty Name "InfoData"}
	InfoData : InfoData_6F19DB2B;
END_STRUCT
END_TYPE

// ---- DUTs/IO/Boxes/EK1122_1FC0878B.TcDUT
{attribute 'GeneratedUsingTerminal: EK1122-0000-0018'}
{attribute addProperty BoxType "EK1122-0000-0018"}
{attribute addProperty Description "EK1122 2 port EtherCAT junction"}
{attribute addProperty Physics "KYKY"}
{attribute addProperty Id "InfoDataAT %I*InfoData_6F19DB2B2"}
{attribute addProperty CRC "532711307"}
{attribute addProperty Size "2"}
TYPE EK1122_1FC0878B EXTENDS EtcSlaveTerminalBase_947E5A46 :
STRUCT
	{attribute addProperty Name "InfoData"}
	InfoData : InfoData_6F19DB2B;
END_STRUCT
END_TYPE

// ---- DUTs/IO/Boxes/ELM3002_B416BFEF.TcDUT
{attribute 'GeneratedUsingTerminal: ELM3002-0000-0016'}
{attribute addProperty BoxType "ELM3002-0000-0016"}
{attribute addProperty Description "ELM3002 2Ch. Ana. Input +/-30V, 24 bit, high precision"}
{attribute addProperty Physics "KK"}
{attribute addProperty Id "PAI_Status_Channel_1AT %I*PAI_Status_Channel_AE4AC1047PAI_Samples_1_Channel_1AT %I*PAI_Samples_1_Channel_EEA517254PAI_Timestamp_Channel_1AT %I*PAI_Timestamp_Channel_6DC4D2968PAI_Status_Channel_2AT %I*PAI_Status_Channel_AE4AC1047PAI_Samples_1_Channel_2AT %I*PAI_Samples_1_Channel_EEA517254WcStateAT %I*WcState_9091E0EB2InfoDataAT %I*InfoData_BEF6B88E18"}
{attribute addProperty CRC "3021389807"}
{attribute addProperty Size "50"}
TYPE ELM3002_B416BFEF EXTENDS EtcSlaveTerminalBase_947E5A46 :
STRUCT
	{attribute addProperty Name "PAI_Status_Channel_1"}
	PAI_Status_Channel_1 : PAI_Status_Channel_AE4AC104;
	{attribute addProperty Name "PAI_Samples_1_Channel_1"}
	PAI_Samples_1_Channel_1 : PAI_Samples_1_Channel_EEA51725;
	{attribute addProperty Name "PAI_Timestamp_Channel_1"}
	PAI_Timestamp_Channel_1 : PAI_Timestamp_Channel_6DC4D296;
	{attribute addProperty Name "PAI_Status_Channel_2"}
	PAI_Status_Channel_2 : PAI_Status_Channel_AE4AC104;
	{attribute addProperty Name "PAI_Samples_1_Channel_2"}
	PAI_Samples_1_Channel_2 : PAI_Samples_1_Channel_EEA51725;
	{attribute addProperty Name "WcState"}
	WcState : WcState_9091E0EB;
	{attribute addProperty Name "InfoData"}
	InfoData : InfoData_BEF6B88E;
END_STRUCT
END_TYPE

// ---- DUTs/IO/Boxes/ELM3004_9E251EA4.TcDUT
{attribute 'GeneratedUsingTerminal: ELM3004-0000-0016'}
{attribute addProperty BoxType "ELM3004-0000-0016"}
{attribute addProperty Description "ELM3004 4Ch. Ana. Input +/-30V, 24 bit, high precision"}
{attribute addProperty Physics "KK"}
{attribute addProperty Id "PAI_Status_Channel_1AT %I*PAI_Status_Channel_AE4AC1047PAI_Samples_1_Channel_1AT %I*PAI_Samples_1_Channel_EEA517254PAI_Timestamp_Channel_1AT %I*PAI_Timestamp_Channel_6DC4D2968PAI_Status_Channel_2AT %I*PAI_Status_Channel_AE4AC1047PAI_Samples_1_Channel_2AT %I*PAI_Samples_1_Channel_EEA517254PAI_Status_Channel_3AT %I*PAI_Status_Channel_AE4AC1047PAI_Samples_1_Channel_3AT %I*PAI_Samples_1_Channel_EEA517254PAI_Status_Channel_4AT %I*PAI_Status_Channel_AE4AC1047PAI_Samples_1_Channel_4AT %I*PAI_Samples_1_Channel_EEA517254WcStateAT %I*WcState_9091E0EB2InfoDataAT %I*InfoData_BEF6B88E18"}
{attribute addProperty CRC "2653232804"}
{attribute addProperty Size "72"}
TYPE ELM3004_9E251EA4 EXTENDS EtcSlaveTerminalBase_947E5A46 :
STRUCT
	{attribute addProperty Name "PAI_Status_Channel_1"}
	PAI_Status_Channel_1 : PAI_Status_Channel_AE4AC104;
	{attribute addProperty Name "PAI_Samples_1_Channel_1"}
	PAI_Samples_1_Channel_1 : PAI_Samples_1_Channel_EEA51725;
	{attribute addProperty Name "PAI_Timestamp_Channel_1"}
	PAI_Timestamp_Channel_1 : PAI_Timestamp_Channel_6DC4D296;
	{attribute addProperty Name "PAI_Status_Channel_2"}
	PAI_Status_Channel_2 : PAI_Status_Channel_AE4AC104;
	{attribute addProperty Name "PAI_Samples_1_Channel_2"}
	PAI_Samples_1_Channel_2 : PAI_Samples_1_Channel_EEA51725;
	{attribute addProperty Name "PAI_Status_Channel_3"}
	PAI_Status_Channel_3 : PAI_Status_Channel_AE4AC104;
	{attribute addProperty Name "PAI_Samples_1_Channel_3"}
	PAI_Samples_1_Channel_3 : PAI_Samples_1_Channel_EEA51725;
	{attribute addProperty Name "PAI_Status_Channel_4"}
	PAI_Status_Channel_4 : PAI_Status_Channel_AE4AC104;
	{attribute addProperty Name "PAI_Samples_1_Channel_4"}
	PAI_Samples_1_Channel_4 : PAI_Samples_1_Channel_EEA51725;
	{attribute addProperty Name "WcState"}
	WcState : WcState_9091E0EB;
	{attribute addProperty Name "InfoData"}
	InfoData : InfoData_BEF6B88E;
END_STRUCT
END_TYPE

// ---- DUTs/IO/Boxes/ELM3102_B416BFEF.TcDUT
{attribute 'GeneratedUsingTerminal: ELM3102-0000-0016'}
{attribute addProperty BoxType "ELM3102-0000-0016"}
{attribute addProperty Description "ELM3102 2Ch. Ana. Input +/-20mA, 24 bit, high precision"}
{attribute addProperty Physics "KK"}
{attribute addProperty Id "PAI_Status_Channel_1AT %I*PAI_Status_Channel_AE4AC1047PAI_Samples_1_Channel_1AT %I*PAI_Samples_1_Channel_EEA517254PAI_Timestamp_Channel_1AT %I*PAI_Timestamp_Channel_6DC4D2968PAI_Status_Channel_2AT %I*PAI_Status_Channel_AE4AC1047PAI_Samples_1_Channel_2AT %I*PAI_Samples_1_Channel_EEA517254WcStateAT %I*WcState_9091E0EB2InfoDataAT %I*InfoData_BEF6B88E18"}
{attribute addProperty CRC "3021389807"}
{attribute addProperty Size "50"}
TYPE ELM3102_B416BFEF EXTENDS EtcSlaveTerminalBase_947E5A46 :
STRUCT
	{attribute addProperty Name "PAI_Status_Channel_1"}
	PAI_Status_Channel_1 : PAI_Status_Channel_AE4AC104;
	{attribute addProperty Name "PAI_Samples_1_Channel_1"}
	PAI_Samples_1_Channel_1 : PAI_Samples_1_Channel_EEA51725;
	{attribute addProperty Name "PAI_Timestamp_Channel_1"}
	PAI_Timestamp_Channel_1 : PAI_Timestamp_Channel_6DC4D296;
	{attribute addProperty Name "PAI_Status_Channel_2"}
	PAI_Status_Channel_2 : PAI_Status_Channel_AE4AC104;
	{attribute addProperty Name "PAI_Samples_1_Channel_2"}
	PAI_Samples_1_Channel_2 : PAI_Samples_1_Channel_EEA51725;
	{attribute addProperty Name "WcState"}
	WcState : WcState_9091E0EB;
	{attribute addProperty Name "InfoData"}
	InfoData : InfoData_BEF6B88E;
END_STRUCT
END_TYPE

// ---- DUTs/IO/Boxes/ELM3104_9E251EA4.TcDUT
{attribute 'GeneratedUsingTerminal: ELM3104-0000-0016'}
{attribute addProperty BoxType "ELM3104-0000-0016"}
{attribute addProperty Description "ELM3104 4Ch. Ana. Input +/-20mA, 24 bit, high precision"}
{attribute addProperty Physics "KK"}
{attribute addProperty Id "PAI_Status_Channel_1AT %I*PAI_Status_Channel_AE4AC1047PAI_Samples_1_Channel_1AT %I*PAI_Samples_1_Channel_EEA517254PAI_Timestamp_Channel_1AT %I*PAI_Timestamp_Channel_6DC4D2968PAI_Status_Channel_2AT %I*PAI_Status_Channel_AE4AC1047PAI_Samples_1_Channel_2AT %I*PAI_Samples_1_Channel_EEA517254PAI_Status_Channel_3AT %I*PAI_Status_Channel_AE4AC1047PAI_Samples_1_Channel_3AT %I*PAI_Samples_1_Channel_EEA517254PAI_Status_Channel_4AT %I*PAI_Status_Channel_AE4AC1047PAI_Samples_1_Channel_4AT %I*PAI_Samples_1_Channel_EEA517254WcStateAT %I*WcState_9091E0EB2InfoDataAT %I*InfoData_BEF6B88E18"}
{attribute addProperty CRC "2653232804"}
{attribute addProperty Size "72"}
TYPE ELM3104_9E251EA4 EXTENDS EtcSlaveTerminalBase_947E5A46 :
STRUCT
	{attribute addProperty Name "PAI_Status_Channel_1"}
	PAI_Status_Channel_1 : PAI_Status_Channel_AE4AC104;
	{attribute addProperty Name "PAI_Samples_1_Channel_1"}
	PAI_Samples_1_Channel_1 : PAI_Samples_1_Channel_EEA51725;
	{attribute addProperty Name "PAI_Timestamp_Channel_1"}
	PAI_Timestamp_Channel_1 : PAI_Timestamp_Channel_6DC4D296;
	{attribute addProperty Name "PAI_Status_Channel_2"}
	PAI_Status_Channel_2 : PAI_Status_Channel_AE4AC104;
	{attribute addProperty Name "PAI_Samples_1_Channel_2"}
	PAI_Samples_1_Channel_2 : PAI_Samples_1_Channel_EEA51725;
	{attribute addProperty Name "PAI_Status_Channel_3"}
	PAI_Status_Channel_3 : PAI_Status_Channel_AE4AC104;
	{attribute addProperty Name "PAI_Samples_1_Channel_3"}
	PAI_Samples_1_Channel_3 : PAI_Samples_1_Channel_EEA51725;
	{attribute addProperty Name "PAI_Status_Channel_4"}
	PAI_Status_Channel_4 : PAI_Status_Channel_AE4AC104;
	{attribute addProperty Name "PAI_Samples_1_Channel_4"}
	PAI_Samples_1_Channel_4 : PAI_Samples_1_Channel_EEA51725;
	{attribute addProperty Name "WcState"}
	WcState : WcState_9091E0EB;
	{attribute addProperty Name "InfoData"}
	InfoData : InfoData_BEF6B88E;
END_STRUCT
END_TYPE

// ---- DUTs/IO/Boxes/ELM3142_B416BFEF.TcDUT
{attribute 'GeneratedUsingTerminal: ELM3142-0000-0016'}
{attribute addProperty BoxType "ELM3142-0000-0016"}
{attribute addProperty Description "ELM3142-0000 2Ch. Ana. Input +/-10V, +/-20mA, 24 bit, high precision"}
{attribute addProperty Physics "KK"}
{attribute addProperty Id "PAI_Status_Channel_1AT %I*PAI_Status_Channel_AE4AC1047PAI_Samples_1_Channel_1AT %I*PAI_Samples_1_Channel_EEA517254PAI_Timestamp_Channel_1AT %I*PAI_Timestamp_Channel_6DC4D2968PAI_Status_Channel_2AT %I*PAI_Status_Channel_AE4AC1047PAI_Samples_1_Channel_2AT %I*PAI_Samples_1_Channel_EEA517254WcStateAT %I*WcState_9091E0EB2InfoDataAT %I*InfoData_BEF6B88E18"}
{attribute addProperty CRC "3021389807"}
{attribute addProperty Size "50"}
TYPE ELM3142_B416BFEF EXTENDS EtcSlaveTerminalBase_947E5A46 :
STRUCT
	{attribute addProperty Name "PAI_Status_Channel_1"}
	PAI_Status_Channel_1 : PAI_Status_Channel_AE4AC104;
	{attribute addProperty Name "PAI_Samples_1_Channel_1"}
	PAI_Samples_1_Channel_1 : PAI_Samples_1_Channel_EEA51725;
	{attribute addProperty Name "PAI_Timestamp_Channel_1"}
	PAI_Timestamp_Channel_1 : PAI_Timestamp_Channel_6DC4D296;
	{attribute addProperty Name "PAI_Status_Channel_2"}
	PAI_Status_Channel_2 : PAI_Status_Channel_AE4AC104;
	{attribute addProperty Name "PAI_Samples_1_Channel_2"}
	PAI_Samples_1_Channel_2 : PAI_Samples_1_Channel_EEA51725;
	{attribute addProperty Name "WcState"}
	WcState : WcState_9091E0EB;
	{attribute addProperty Name "InfoData"}
	InfoData : InfoData_BEF6B88E;
END_STRUCT
END_TYPE

// ---- DUTs/IO/Boxes/ELM3144_9E251EA4.TcDUT
{attribute 'GeneratedUsingTerminal: ELM3144-0000-0016'}
{attribute addProperty BoxType "ELM3144-0000-0016"}
{attribute addProperty Description "ELM3144-0000 4Ch. Ana. Input +/-10V, +/-20mA, 24 bit, high precision"}
{attribute addProperty Physics "KK"}
{attribute addProperty Id "PAI_Status_Channel_1AT %I*PAI_Status_Channel_AE4AC1047PAI_Samples_1_Channel_1AT %I*PAI_Samples_1_Channel_EEA517254PAI_Timestamp_Channel_1AT %I*PAI_Timestamp_Channel_6DC4D2968PAI_Status_Channel_2AT %I*PAI_Status_Channel_AE4AC1047PAI_Samples_1_Channel_2AT %I*PAI_Samples_1_Channel_EEA517254PAI_Status_Channel_3AT %I*PAI_Status_Channel_AE4AC1047PAI_Samples_1_Channel_3AT %I*PAI_Samples_1_Channel_EEA517254PAI_Status_Channel_4AT %I*PAI_Status_Channel_AE4AC1047PAI_Samples_1_Channel_4AT %I*PAI_Samples_1_Channel_EEA517254WcStateAT %I*WcState_9091E0EB2InfoDataAT %I*InfoData_BEF6B88E18"}
{attribute addProperty CRC "2653232804"}
{attribute addProperty Size "72"}
TYPE ELM3144_9E251EA4 EXTENDS EtcSlaveTerminalBase_947E5A46 :
STRUCT
	{attribute addProperty Name "PAI_Status_Channel_1"}
	PAI_Status_Channel_1 : PAI_Status_Channel_AE4AC104;
	{attribute addProperty Name "PAI_Samples_1_Channel_1"}
	PAI_Samples_1_Channel_1 : PAI_Samples_1_Channel_EEA51725;
	{attribute addProperty Name "PAI_Timestamp_Channel_1"}
	PAI_Timestamp_Channel_1 : PAI_Timestamp_Channel_6DC4D296;
	{attribute addProperty Name "PAI_Status_Channel_2"}
	PAI_Status_Channel_2 : PAI_Status_Channel_AE4AC104;
	{attribute addProperty Name "PAI_Samples_1_Channel_2"}
	PAI_Samples_1_Channel_2 : PAI_Samples_1_Channel_EEA51725;
	{attribute addProperty Name "PAI_Status_Channel_3"}
	PAI_Status_Channel_3 : PAI_Status_Channel_AE4AC104;
	{attribute addProperty Name "PAI_Samples_1_Channel_3"}
	PAI_Samples_1_Channel_3 : PAI_Samples_1_Channel_EEA51725;
	{attribute addProperty Name "PAI_Status_Channel_4"}
	PAI_Status_Channel_4 : PAI_Status_Channel_AE4AC104;
	{attribute addProperty Name "PAI_Samples_1_Channel_4"}
	PAI_Samples_1_Channel_4 : PAI_Samples_1_Channel_EEA51725;
	{attribute addProperty Name "WcState"}
	WcState : WcState_9091E0EB;
	{attribute addProperty Name "InfoData"}
	InfoData : InfoData_BEF6B88E;
END_STRUCT
END_TYPE

// ---- DUTs/IO/Boxes/ELM3146_EA6DB5D7.TcDUT
{attribute 'GeneratedUsingTerminal: ELM3146-0000-0016'}
{attribute addProperty BoxType "ELM3146-0000-0016"}
{attribute addProperty Description "ELM3146-0000 6Ch. Ana. Input +/-10V, +/-20mA, 24 bit, high precision"}
{attribute addProperty Physics "KK"}
{attribute addProperty Id "PAI_Status_Channel_1AT %I*PAI_Status_Channel_AE4AC1047PAI_Samples_1_Channel_1AT %I*PAI_Samples_1_Channel_EEA517254PAI_Timestamp_Channel_1AT %I*PAI_Timestamp_Channel_6DC4D2968PAI_Status_Channel_2AT %I*PAI_Status_Channel_AE4AC1047PAI_Samples_1_Channel_2AT %I*PAI_Samples_1_Channel_EEA517254PAI_Status_Channel_3AT %I*PAI_Status_Channel_AE4AC1047PAI_Samples_1_Channel_3AT %I*PAI_Samples_1_Channel_EEA517254PAI_Status_Channel_4AT %I*PAI_Status_Channel_AE4AC1047PAI_Samples_1_Channel_4AT %I*PAI_Samples_1_Channel_EEA517254PAI_Status_Channel_5AT %I*PAI_Status_Channel_AE4AC1047PAI_Samples_1_Channel_5AT %I*PAI_Samples_1_Channel_EEA517254PAI_Status_Channel_6AT %I*PAI_Status_Channel_AE4AC1047PAI_Samples_1_Channel_6AT %I*PAI_Samples_1_Channel_EEA517254WcStateAT %I*WcState_9091E0EB2InfoDataAT %I*InfoData_BEF6B88E18"}
{attribute addProperty CRC "3933058519"}
{attribute addProperty Size "94"}
TYPE ELM3146_EA6DB5D7 EXTENDS EtcSlaveTerminalBase_947E5A46 :
STRUCT
	{attribute addProperty Name "PAI_Status_Channel_1"}
	PAI_Status_Channel_1 : PAI_Status_Channel_AE4AC104;
	{attribute addProperty Name "PAI_Samples_1_Channel_1"}
	PAI_Samples_1_Channel_1 : PAI_Samples_1_Channel_EEA51725;
	{attribute addProperty Name "PAI_Timestamp_Channel_1"}
	PAI_Timestamp_Channel_1 : PAI_Timestamp_Channel_6DC4D296;
	{attribute addProperty Name "PAI_Status_Channel_2"}
	PAI_Status_Channel_2 : PAI_Status_Channel_AE4AC104;
	{attribute addProperty Name "PAI_Samples_1_Channel_2"}
	PAI_Samples_1_Channel_2 : PAI_Samples_1_Channel_EEA51725;
	{attribute addProperty Name "PAI_Status_Channel_3"}
	PAI_Status_Channel_3 : PAI_Status_Channel_AE4AC104;
	{attribute addProperty Name "PAI_Samples_1_Channel_3"}
	PAI_Samples_1_Channel_3 : PAI_Samples_1_Channel_EEA51725;
	{attribute addProperty Name "PAI_Status_Channel_4"}
	PAI_Status_Channel_4 : PAI_Status_Channel_AE4AC104;
	{attribute addProperty Name "PAI_Samples_1_Channel_4"}
	PAI_Samples_1_Channel_4 : PAI_Samples_1_Channel_EEA51725;
	{attribute addProperty Name "PAI_Status_Channel_5"}
	PAI_Status_Channel_5 : PAI_Status_Channel_AE4AC104;
	{attribute addProperty Name "PAI_Samples_1_Channel_5"}
	PAI_Samples_1_Channel_5 : PAI_Samples_1_Channel_EEA51725;
	{attribute addProperty Name "PAI_Status_Channel_6"}
	PAI_Status_Channel_6 : PAI_Status_Channel_AE4AC104;
	{attribute addProperty Name "PAI_Samples_1_Channel_6"}
	PAI_Samples_1_Channel_6 : PAI_Samples_1_Channel_EEA51725;
	{attribute addProperty Name "WcState"}
	WcState : WcState_9091E0EB;
	{attribute addProperty Name "InfoData"}
	InfoData : InfoData_BEF6B88E;
END_STRUCT
END_TYPE

// ---- DUTs/IO/Boxes/ELM3148_0838C628.TcDUT
{attribute 'GeneratedUsingTerminal: ELM3148-0000-0017'}
{attribute addProperty BoxType "ELM3148-0000-0017"}
{attribute addProperty Description "ELM3148-0000 8Ch. Ana. Input +/-10V, +/-20mA, 24 bit, high precision"}
{attribute addProperty Physics "KK"}
{attribute addProperty Id "PAI_Status_Channel_1AT %I*PAI_Status_Channel_AE4AC1047PAI_Samples_1_Channel_1AT %I*PAI_Samples_1_Channel_EEA517254PAI_Timestamp_Channel_1AT %I*PAI_Timestamp_Channel_6DC4D2968PAI_Status_Channel_2AT %I*PAI_Status_Channel_AE4AC1047PAI_Samples_1_Channel_2AT %I*PAI_Samples_1_Channel_EEA517254PAI_Status_Channel_3AT %I*PAI_Status_Channel_AE4AC1047PAI_Samples_1_Channel_3AT %I*PAI_Samples_1_Channel_EEA517254PAI_Status_Channel_4AT %I*PAI_Status_Channel_AE4AC1047PAI_Samples_1_Channel_4AT %I*PAI_Samples_1_Channel_EEA517254PAI_Status_Channel_5AT %I*PAI_Status_Channel_AE4AC1047PAI_Samples_1_Channel_5AT %I*PAI_Samples_1_Channel_EEA517254PAI_Status_Channel_6AT %I*PAI_Status_Channel_AE4AC1047PAI_Samples_1_Channel_6AT %I*PAI_Samples_1_Channel_EEA517254PAI_Status_Channel_7AT %I*PAI_Status_Channel_AE4AC1047PAI_Samples_1_Channel_7AT %I*PAI_Samples_1_Channel_EEA517254PAI_Status_Channel_8AT %I*PAI_Status_Channel_AE4AC1047PAI_Samples_1_Channel_8AT %I*PAI_Samples_1_Channel_EEA517254WcStateAT %I*WcState_9091E0EB2InfoDataAT %I*InfoData_BEF6B88E18"}
{attribute addProperty CRC "137938472"}
{attribute addProperty Size "116"}
TYPE ELM3148_0838C628 EXTENDS EtcSlaveTerminalBase_947E5A46 :
STRUCT
	{attribute addProperty Name "PAI_Status_Channel_1"}
	PAI_Status_Channel_1 : PAI_Status_Channel_AE4AC104;
	{attribute addProperty Name "PAI_Samples_1_Channel_1"}
	PAI_Samples_1_Channel_1 : PAI_Samples_1_Channel_EEA51725;
	{attribute addProperty Name "PAI_Timestamp_Channel_1"}
	PAI_Timestamp_Channel_1 : PAI_Timestamp_Channel_6DC4D296;
	{attribute addProperty Name "PAI_Status_Channel_2"}
	PAI_Status_Channel_2 : PAI_Status_Channel_AE4AC104;
	{attribute addProperty Name "PAI_Samples_1_Channel_2"}
	PAI_Samples_1_Channel_2 : PAI_Samples_1_Channel_EEA51725;
	{attribute addProperty Name "PAI_Status_Channel_3"}
	PAI_Status_Channel_3 : PAI_Status_Channel_AE4AC104;
	{attribute addProperty Name "PAI_Samples_1_Channel_3"}
	PAI_Samples_1_Channel_3 : PAI_Samples_1_Channel_EEA51725;
	{attribute addProperty Name "PAI_Status_Channel_4"}
	PAI_Status_Channel_4 : PAI_Status_Channel_AE4AC104;
	{attribute addProperty Name "PAI_Samples_1_Channel_4"}
	PAI_Samples_1_Channel_4 : PAI_Samples_1_Channel_EEA51725;
	{attribute addProperty Name "PAI_Status_Channel_5"}
	PAI_Status_Channel_5 : PAI_Status_Channel_AE4AC104;
	{attribute addProperty Name "PAI_Samples_1_Channel_5"}
	PAI_Samples_1_Channel_5 : PAI_Samples_1_Channel_EEA51725;
	{attribute addProperty Name "PAI_Status_Channel_6"}
	PAI_Status_Channel_6 : PAI_Status_Channel_AE4AC104;
	{attribute addProperty Name "PAI_Samples_1_Channel_6"}
	PAI_Samples_1_Channel_6 : PAI_Samples_1_Channel_EEA51725;
	{attribute addProperty Name "PAI_Status_Channel_7"}
	PAI_Status_Channel_7 : PAI_Status_Channel_AE4AC104;
	{attribute addProperty Name "PAI_Samples_1_Channel_7"}
	PAI_Samples_1_Channel_7 : PAI_Samples_1_Channel_EEA51725;
	{attribute addProperty Name "PAI_Status_Channel_8"}
	PAI_Status_Channel_8 : PAI_Status_Channel_AE4AC104;
	{attribute addProperty Name "PAI_Samples_1_Channel_8"}
	PAI_Samples_1_Channel_8 : PAI_Samples_1_Channel_EEA51725;
	{attribute addProperty Name "WcState"}
	WcState : WcState_9091E0EB;
	{attribute addProperty Name "InfoData"}
	InfoData : InfoData_BEF6B88E;
END_STRUCT
END_TYPE

// ---- DUTs/IO/Boxes/ELM3502_B416BFEF.TcDUT
{attribute 'GeneratedUsingTerminal: ELM3502-0000-0016'}
{attribute addProperty BoxType "ELM3502-0000-0016"}
{attribute addProperty Description "ELM3502-0000 2Ch. Bridge Measuring (SG), 24 bit, high precision"}
{attribute addProperty Physics "KK"}
{attribute addProperty Id "PAI_Status_Channel_1AT %I*PAI_Status_Channel_AE4AC1047PAI_Samples_1_Channel_1AT %I*PAI_Samples_1_Channel_EEA517254PAI_Timestamp_Channel_1AT %I*PAI_Timestamp_Channel_6DC4D2968PAI_Status_Channel_2AT %I*PAI_Status_Channel_AE4AC1047PAI_Samples_1_Channel_2AT %I*PAI_Samples_1_Channel_EEA517254WcStateAT %I*WcState_9091E0EB2InfoDataAT %I*InfoData_BEF6B88E18"}
{attribute addProperty CRC "3021389807"}
{attribute addProperty Size "50"}
TYPE ELM3502_B416BFEF EXTENDS EtcSlaveTerminalBase_947E5A46 :
STRUCT
	{attribute addProperty Name "PAI_Status_Channel_1"}
	PAI_Status_Channel_1 : PAI_Status_Channel_AE4AC104;
	{attribute addProperty Name "PAI_Samples_1_Channel_1"}
	PAI_Samples_1_Channel_1 : PAI_Samples_1_Channel_EEA51725;
	{attribute addProperty Name "PAI_Timestamp_Channel_1"}
	PAI_Timestamp_Channel_1 : PAI_Timestamp_Channel_6DC4D296;
	{attribute addProperty Name "PAI_Status_Channel_2"}
	PAI_Status_Channel_2 : PAI_Status_Channel_AE4AC104;
	{attribute addProperty Name "PAI_Samples_1_Channel_2"}
	PAI_Samples_1_Channel_2 : PAI_Samples_1_Channel_EEA51725;
	{attribute addProperty Name "WcState"}
	WcState : WcState_9091E0EB;
	{attribute addProperty Name "InfoData"}
	InfoData : InfoData_BEF6B88E;
END_STRUCT
END_TYPE

// ---- DUTs/IO/Boxes/ELM3504_9E251EA4.TcDUT
{attribute 'GeneratedUsingTerminal: ELM3504-0000-0016'}
{attribute addProperty BoxType "ELM3504-0000-0016"}
{attribute addProperty Description "ELM3504-0000 4Ch. Bridge Measuring (SG), 24 bit, high precision"}
{attribute addProperty Physics "KK"}
{attribute addProperty Id "PAI_Status_Channel_1AT %I*PAI_Status_Channel_AE4AC1047PAI_Samples_1_Channel_1AT %I*PAI_Samples_1_Channel_EEA517254PAI_Timestamp_Channel_1AT %I*PAI_Timestamp_Channel_6DC4D2968PAI_Status_Channel_2AT %I*PAI_Status_Channel_AE4AC1047PAI_Samples_1_Channel_2AT %I*PAI_Samples_1_Channel_EEA517254PAI_Status_Channel_3AT %I*PAI_Status_Channel_AE4AC1047PAI_Samples_1_Channel_3AT %I*PAI_Samples_1_Channel_EEA517254PAI_Status_Channel_4AT %I*PAI_Status_Channel_AE4AC1047PAI_Samples_1_Channel_4AT %I*PAI_Samples_1_Channel_EEA517254WcStateAT %I*WcState_9091E0EB2InfoDataAT %I*InfoData_BEF6B88E18"}
{attribute addProperty CRC "2653232804"}
{attribute addProperty Size "72"}
TYPE ELM3504_9E251EA4 EXTENDS EtcSlaveTerminalBase_947E5A46 :
STRUCT
	{attribute addProperty Name "PAI_Status_Channel_1"}
	PAI_Status_Channel_1 : PAI_Status_Channel_AE4AC104;
	{attribute addProperty Name "PAI_Samples_1_Channel_1"}
	PAI_Samples_1_Channel_1 : PAI_Samples_1_Channel_EEA51725;
	{attribute addProperty Name "PAI_Timestamp_Channel_1"}
	PAI_Timestamp_Channel_1 : PAI_Timestamp_Channel_6DC4D296;
	{attribute addProperty Name "PAI_Status_Channel_2"}
	PAI_Status_Channel_2 : PAI_Status_Channel_AE4AC104;
	{attribute addProperty Name "PAI_Samples_1_Channel_2"}
	PAI_Samples_1_Channel_2 : PAI_Samples_1_Channel_EEA51725;
	{attribute addProperty Name "PAI_Status_Channel_3"}
	PAI_Status_Channel_3 : PAI_Status_Channel_AE4AC104;
	{attribute addProperty Name "PAI_Samples_1_Channel_3"}
	PAI_Samples_1_Channel_3 : PAI_Samples_1_Channel_EEA51725;
	{attribute addProperty Name "PAI_Status_Channel_4"}
	PAI_Status_Channel_4 : PAI_Status_Channel_AE4AC104;
	{attribute addProperty Name "PAI_Samples_1_Channel_4"}
	PAI_Samples_1_Channel_4 : PAI_Samples_1_Channel_EEA51725;
	{attribute addProperty Name "WcState"}
	WcState : WcState_9091E0EB;
	{attribute addProperty Name "InfoData"}
	InfoData : InfoData_BEF6B88E;
END_STRUCT
END_TYPE

// ---- DUTs/IO/Boxes/ELM3602_B416BFEF.TcDUT
{attribute 'GeneratedUsingTerminal: ELM3602-0000-0017'}
{attribute addProperty BoxType "ELM3602-0000-0017"}
{attribute addProperty Description "ELM3602-0000 2Ch. IEPE Sensor, 24 bit, high precision"}
{attribute addProperty Physics "KK"}
{attribute addProperty Id "PAI_Status_Channel_1AT %I*PAI_Status_Channel_AE4AC1047PAI_Samples_1_Channel_1AT %I*PAI_Samples_1_Channel_EEA517254PAI_Timestamp_Channel_1AT %I*PAI_Timestamp_Channel_6DC4D2968PAI_Status_Channel_2AT %I*PAI_Status_Channel_AE4AC1047PAI_Samples_1_Channel_2AT %I*PAI_Samples_1_Channel_EEA517254WcStateAT %I*WcState_9091E0EB2InfoDataAT %I*InfoData_BEF6B88E18"}
{attribute addProperty CRC "3021389807"}
{attribute addProperty Size "50"}
TYPE ELM3602_B416BFEF EXTENDS EtcSlaveTerminalBase_947E5A46 :
STRUCT
	{attribute addProperty Name "PAI_Status_Channel_1"}
	PAI_Status_Channel_1 : PAI_Status_Channel_AE4AC104;
	{attribute addProperty Name "PAI_Samples_1_Channel_1"}
	PAI_Samples_1_Channel_1 : PAI_Samples_1_Channel_EEA51725;
	{attribute addProperty Name "PAI_Timestamp_Channel_1"}
	PAI_Timestamp_Channel_1 : PAI_Timestamp_Channel_6DC4D296;
	{attribute addProperty Name "PAI_Status_Channel_2"}
	PAI_Status_Channel_2 : PAI_Status_Channel_AE4AC104;
	{attribute addProperty Name "PAI_Samples_1_Channel_2"}
	PAI_Samples_1_Channel_2 : PAI_Samples_1_Channel_EEA51725;
	{attribute addProperty Name "WcState"}
	WcState : WcState_9091E0EB;
	{attribute addProperty Name "InfoData"}
	InfoData : InfoData_BEF6B88E;
END_STRUCT
END_TYPE

// ---- DUTs/IO/Boxes/ELM3604_9E251EA4.TcDUT
{attribute 'GeneratedUsingTerminal: ELM3604-0000-0017'}
{attribute addProperty BoxType "ELM3604-0000-0017"}
{attribute addProperty Description "ELM3604-0000 4Ch. IEPE Sensor, 24 bit, high precision"}
{attribute addProperty Physics "KK"}
{attribute addProperty Id "PAI_Status_Channel_1AT %I*PAI_Status_Channel_AE4AC1047PAI_Samples_1_Channel_1AT %I*PAI_Samples_1_Channel_EEA517254PAI_Timestamp_Channel_1AT %I*PAI_Timestamp_Channel_6DC4D2968PAI_Status_Channel_2AT %I*PAI_Status_Channel_AE4AC1047PAI_Samples_1_Channel_2AT %I*PAI_Samples_1_Channel_EEA517254PAI_Status_Channel_3AT %I*PAI_Status_Channel_AE4AC1047PAI_Samples_1_Channel_3AT %I*PAI_Samples_1_Channel_EEA517254PAI_Status_Channel_4AT %I*PAI_Status_Channel_AE4AC1047PAI_Samples_1_Channel_4AT %I*PAI_Samples_1_Channel_EEA517254WcStateAT %I*WcState_9091E0EB2InfoDataAT %I*InfoData_BEF6B88E18"}
{attribute addProperty CRC "2653232804"}
{attribute addProperty Size "72"}
TYPE ELM3604_9E251EA4 EXTENDS EtcSlaveTerminalBase_947E5A46 :
STRUCT
	{attribute addProperty Name "PAI_Status_Channel_1"}
	PAI_Status_Channel_1 : PAI_Status_Channel_AE4AC104;
	{attribute addProperty Name "PAI_Samples_1_Channel_1"}
	PAI_Samples_1_Channel_1 : PAI_Samples_1_Channel_EEA51725;
	{attribute addProperty Name "PAI_Timestamp_Channel_1"}
	PAI_Timestamp_Channel_1 : PAI_Timestamp_Channel_6DC4D296;
	{attribute addProperty Name "PAI_Status_Channel_2"}
	PAI_Status_Channel_2 : PAI_Status_Channel_AE4AC104;
	{attribute addProperty Name "PAI_Samples_1_Channel_2"}
	PAI_Samples_1_Channel_2 : PAI_Samples_1_Channel_EEA51725;
	{attribute addProperty Name "PAI_Status_Channel_3"}
	PAI_Status_Channel_3 : PAI_Status_Channel_AE4AC104;
	{attribute addProperty Name "PAI_Samples_1_Channel_3"}
	PAI_Samples_1_Channel_3 : PAI_Samples_1_Channel_EEA51725;
	{attribute addProperty Name "PAI_Status_Channel_4"}
	PAI_Status_Channel_4 : PAI_Status_Channel_AE4AC104;
	{attribute addProperty Name "PAI_Samples_1_Channel_4"}
	PAI_Samples_1_Channel_4 : PAI_Samples_1_Channel_EEA51725;
	{attribute addProperty Name "WcState"}
	WcState : WcState_9091E0EB;
	{attribute addProperty Name "InfoData"}
	InfoData : InfoData_BEF6B88E;
END_STRUCT
END_TYPE

// ---- DUTs/IO/Boxes/ELM3702_B416BFEF.TcDUT
{attribute 'GeneratedUsingTerminal: ELM3702-0000-0016'}
{attribute addProperty BoxType "ELM3702-0000-0016"}
{attribute addProperty Description "ELM3702-0000 2Ch. Ana. Input +/-60V, +/-20mA, TC, RTD, Bridge Measuring (SG), IEPE, 24 bit, high precision"}
{attribute addProperty Physics "KK"}
{attribute addProperty Id "PAI_Status_Channel_1AT %I*PAI_Status_Channel_AE4AC1047PAI_Samples_1_Channel_1AT %I*PAI_Samples_1_Channel_EEA517254PAI_Timestamp_Channel_1AT %I*PAI_Timestamp_Channel_6DC4D2968PAI_Status_Channel_2AT %I*PAI_Status_Channel_AE4AC1047PAI_Samples_1_Channel_2AT %I*PAI_Samples_1_Channel_EEA517254WcStateAT %I*WcState_9091E0EB2InfoDataAT %I*InfoData_BEF6B88E18"}
{attribute addProperty CRC "3021389807"}
{attribute addProperty Size "50"}
TYPE ELM3702_B416BFEF EXTENDS EtcSlaveTerminalBase_947E5A46 :
STRUCT
	{attribute addProperty Name "PAI_Status_Channel_1"}
	PAI_Status_Channel_1 : PAI_Status_Channel_AE4AC104;
	{attribute addProperty Name "PAI_Samples_1_Channel_1"}
	PAI_Samples_1_Channel_1 : PAI_Samples_1_Channel_EEA51725;
	{attribute addProperty Name "PAI_Timestamp_Channel_1"}
	PAI_Timestamp_Channel_1 : PAI_Timestamp_Channel_6DC4D296;
	{attribute addProperty Name "PAI_Status_Channel_2"}
	PAI_Status_Channel_2 : PAI_Status_Channel_AE4AC104;
	{attribute addProperty Name "PAI_Samples_1_Channel_2"}
	PAI_Samples_1_Channel_2 : PAI_Samples_1_Channel_EEA51725;
	{attribute addProperty Name "WcState"}
	WcState : WcState_9091E0EB;
	{attribute addProperty Name "InfoData"}
	InfoData : InfoData_BEF6B88E;
END_STRUCT
END_TYPE

// ---- DUTs/IO/Boxes/ELM3704_9E251EA4.TcDUT
{attribute 'GeneratedUsingTerminal: ELM3704-0000-0016'}
{attribute addProperty BoxType "ELM3704-0000-0016"}
{attribute addProperty Description "ELM3704-0000 4Ch. Ana. Input +/-60V, +/-20mA, TC, RTD, Bridge Measuring (SG), IEPE, 24 bit, high precision"}
{attribute addProperty Physics "KK"}
{attribute addProperty Id "PAI_Status_Channel_1AT %I*PAI_Status_Channel_AE4AC1047PAI_Samples_1_Channel_1AT %I*PAI_Samples_1_Channel_EEA517254PAI_Timestamp_Channel_1AT %I*PAI_Timestamp_Channel_6DC4D2968PAI_Status_Channel_2AT %I*PAI_Status_Channel_AE4AC1047PAI_Samples_1_Channel_2AT %I*PAI_Samples_1_Channel_EEA517254PAI_Status_Channel_3AT %I*PAI_Status_Channel_AE4AC1047PAI_Samples_1_Channel_3AT %I*PAI_Samples_1_Channel_EEA517254PAI_Status_Channel_4AT %I*PAI_Status_Channel_AE4AC1047PAI_Samples_1_Channel_4AT %I*PAI_Samples_1_Channel_EEA517254WcStateAT %I*WcState_9091E0EB2InfoDataAT %I*InfoData_BEF6B88E18"}
{attribute addProperty CRC "2653232804"}
{attribute addProperty Size "72"}
TYPE ELM3704_9E251EA4 EXTENDS EtcSlaveTerminalBase_947E5A46 :
STRUCT
	{attribute addProperty Name "PAI_Status_Channel_1"}
	PAI_Status_Channel_1 : PAI_Status_Channel_AE4AC104;
	{attribute addProperty Name "PAI_Samples_1_Channel_1"}
	PAI_Samples_1_Channel_1 : PAI_Samples_1_Channel_EEA51725;
	{attribute addProperty Name "PAI_Timestamp_Channel_1"}
	PAI_Timestamp_Channel_1 : PAI_Timestamp_Channel_6DC4D296;
	{attribute addProperty Name "PAI_Status_Channel_2"}
	PAI_Status_Channel_2 : PAI_Status_Channel_AE4AC104;
	{attribute addProperty Name "PAI_Samples_1_Channel_2"}
	PAI_Samples_1_Channel_2 : PAI_Samples_1_Channel_EEA51725;
	{attribute addProperty Name "PAI_Status_Channel_3"}
	PAI_Status_Channel_3 : PAI_Status_Channel_AE4AC104;
	{attribute addProperty Name "PAI_Samples_1_Channel_3"}
	PAI_Samples_1_Channel_3 : PAI_Samples_1_Channel_EEA51725;
	{attribute addProperty Name "PAI_Status_Channel_4"}
	PAI_Status_Channel_4 : PAI_Status_Channel_AE4AC104;
	{attribute addProperty Name "PAI_Samples_1_Channel_4"}
	PAI_Samples_1_Channel_4 : PAI_Samples_1_Channel_EEA51725;
	{attribute addProperty Name "WcState"}
	WcState : WcState_9091E0EB;
	{attribute addProperty Name "InfoData"}
	InfoData : InfoData_BEF6B88E;
END_STRUCT
END_TYPE

// ---- DUTs/IO/Boxes/ELM9410_DD553935.TcDUT
{attribute 'GeneratedUsingTerminal: ELM9410-0000-0016'}
{attribute addProperty BoxType "ELM9410-0000-0016"}
{attribute addProperty Description "ELM9410 E-Bus Power Supplier (Diagnostics, isolated)"}
{attribute addProperty Physics "KK"}
{attribute addProperty Id "MMS_Device_InputsAT %I*MMS_Device_Inputs_7D6F87344MMS_Acceleration_StatusAT %I*MMS_Acceleration_Status_117690999MMS_Acceleration_X_AxisAT %I*MMS_Acceleration_X_Axis_80E77D6A2MMS_Acceleration_Y_AxisAT %I*MMS_Acceleration_Y_Axis_80E77D6A2MMS_Acceleration_Z_AxisAT %I*MMS_Acceleration_Z_Axis_80E77D6A2MMS_Acceleration_TimestampAT %I*MMS_Acceleration_Timestamp_8B9FE1A28MMS_Voltage_Us_In_InputsAT %I*MMS_Voltage_Us_In_Inputs_60D55C7211MMS_Voltage_Up_In_InputsAT %I*MMS_Voltage_Up_In_Inputs_60D55C7211MMS_Voltage_Up_Out_InputsAT %I*MMS_Voltage_Up_Out_Inputs_60D55C7211MMS_Device_OutputsAT %Q*MMS_Device_Outputs_E6E6F9D11WcStateAT %I*WcState_9091E0EB2InfoDataAT %I*InfoData_BEF6B88E18"}
{attribute addProperty CRC "3713349941"}
{attribute addProperty Size "81"}
TYPE ELM9410_DD553935 EXTENDS EtcSlaveTerminalBase_947E5A46 :
STRUCT
	{attribute addProperty Name "MMS_Device_Inputs"}
	MMS_Device_Inputs : MMS_Device_Inputs_7D6F8734;
	{attribute addProperty Name "MMS_Acceleration_Status"}
	MMS_Acceleration_Status : MMS_Acceleration_Status_11769099;
	{attribute addProperty Name "MMS_Acceleration_X_Axis"}
	MMS_Acceleration_X_Axis : MMS_Acceleration_X_Axis_80E77D6A;
	{attribute addProperty Name "MMS_Acceleration_Y_Axis"}
	MMS_Acceleration_Y_Axis : MMS_Acceleration_Y_Axis_80E77D6A;
	{attribute addProperty Name "MMS_Acceleration_Z_Axis"}
	MMS_Acceleration_Z_Axis : MMS_Acceleration_Z_Axis_80E77D6A;
	{attribute addProperty Name "MMS_Acceleration_Timestamp"}
	MMS_Acceleration_Timestamp : MMS_Acceleration_Timestamp_8B9FE1A2;
	{attribute addProperty Name "MMS_Voltage_Us_In_Inputs"}
	MMS_Voltage_Us_In_Inputs : MMS_Voltage_Us_In_Inputs_60D55C72;
	{attribute addProperty Name "MMS_Voltage_Up_In_Inputs"}
	MMS_Voltage_Up_In_Inputs : MMS_Voltage_Up_In_Inputs_60D55C72;
	{attribute addProperty Name "MMS_Voltage_Up_Out_Inputs"}
	MMS_Voltage_Up_Out_Inputs : MMS_Voltage_Up_Out_Inputs_60D55C72;
	{attribute addProperty Name "MMS_Device_Outputs"}
	MMS_Device_Outputs : MMS_Device_Outputs_E6E6F9D1;
	{attribute addProperty Name "WcState"}
	WcState : WcState_9091E0EB;
	{attribute addProperty Name "InfoData"}
	InfoData : InfoData_BEF6B88E;
END_STRUCT
END_TYPE

// ---- DUTs/IO/Devices/SyncUnitTask_2D604ED5.TcDUT
{attribute 'GeneratedUsingTerminal: IODEVICETYPE_ETHERCATPROT'}
{attribute addProperty BoxType "IODEVICETYPE_ETHERCATPROT"}
{attribute addProperty Id "WcStateAT %I*WcState_0B2B16F91InfoDataAT %I*InfoData_2A97D6CF8"}
{attribute addProperty CRC "761286357"}
{attribute addProperty Size "9"}
TYPE SyncUnitTask_2D604ED5 :
STRUCT
	{attribute addProperty Name "WcState"}
	WcState : WcState_0B2B16F9;
	{attribute addProperty Name "InfoData"}
	InfoData : InfoData_2A97D6CF;
END_STRUCT
END_TYPE

// ---- DUTs/IO/Devices/SyncUnitTasks_6FEB8257.TcDUT
{attribute 'GeneratedUsingTerminal: '}
{attribute addProperty BoxType ""}
{attribute addProperty Id "unreferencedAT %I*SyncUnitTask_2D604ED59PlcTaskAT %I*SyncUnitTask_2D604ED59"}
{attribute addProperty CRC "1877705303"}
{attribute addProperty Size "18"}
TYPE SyncUnitTasks_6FEB8257 :
STRUCT
	{attribute addProperty Name "unreferenced"}
	unreferenced : SyncUnitTask_2D604ED5;
	{attribute addProperty Name "PlcTask"}
	PlcTask : SyncUnitTask_2D604ED5;
END_STRUCT
END_TYPE

// ---- DUTs/IO/Devices/SyncUnits_99E584AF.TcDUT
{attribute 'GeneratedUsingTerminal: '}
{attribute addProperty BoxType ""}
{attribute addProperty Id "_defaultAT %I*SyncUnitTasks_6FEB825718"}
{attribute addProperty CRC "2581955759"}
{attribute addProperty Size "18"}
TYPE SyncUnits_99E584AF :
STRUCT
	{attribute addProperty Name "_default"}
	_default : SyncUnitTasks_6FEB8257;
END_STRUCT
END_TYPE

// ---- DUTs/IO/Topology/Beckhoff_ELM3xxxEK1122_1A0BF035.TcDUT
{attribute 'GeneratedUsingTerminal: EK1122-0000-0018'}
{attribute addProperty BoxType "EK1122-0000-0018"}
{attribute addProperty Id "Beckhoff_ELM3xxxsub_EK1100EK1100_1FC0878B2"}
{attribute addProperty CRC "436990005"}
{attribute addProperty Size "2"}
{attribute addProperty Name "Beckhoff ELM3xxxEK1122"}
TYPE Beckhoff_ELM3xxxEK1122_1A0BF035 EXTENDS EK1122_1FC0878B :
STRUCT
	{attribute addProperty Name "Beckhoff ELM3xxxsub EK1100"}
	{attribute addProperty PreviousPort "Beckhoff ELM3xxxEK1122 : D"}
	Beckhoff_ELM3xxxsub_EK1100 : EK1100_1FC0878B;
END_STRUCT
END_TYPE

// ---- DUTs/IO/Topology/Beckhoff_ELM3xxx_31A44528.TcDUT
{attribute 'GeneratedUsingTerminal: EK1100-0000-0018'}
{attribute addProperty BoxType "EK1100-0000-0018"}
{attribute addProperty Id "Beckhoff_ELM3xxxEK1122Beckhoff_ELM3xxxEK1122_1A0BF0352A_0001_ELM3002_0000_0016ELM3002_B416BFEF50A_0002_ELM3002_0000_0017ELM3002_B416BFEF50A_0003_ELM3002_0000_0018ELM3002_B416BFEF50A_0004_ELM3004_0000_0016ELM3004_9E251EA472A_0005_ELM3004_0000_0017ELM3004_9E251EA472A_0006_ELM3004_0000_0018ELM3004_9E251EA472A_0007_ELM3004_0000_0019ELM3004_9E251EA472"}
{attribute addProperty CRC "832849192"}
{attribute addProperty Size "440"}
{attribute addProperty Name "Beckhoff ELM3xxx"}
TYPE Beckhoff_ELM3xxx_31A44528 EXTENDS EK1100_1FC0878B :
STRUCT
	{attribute addProperty Name "Beckhoff ELM3xxxEK1122"}
	{attribute addProperty PreviousPort "Beckhoff ELM3xxx : B"}
	Beckhoff_ELM3xxxEK1122 : Beckhoff_ELM3xxxEK1122_1A0BF035;
	{attribute addProperty Name "A_0001(ELM3002-0000-0016)"}
	{attribute addProperty PreviousPort "Beckhoff ELM3xxxEK1122 : C"}
	A_0001_ELM3002_0000_0016 : ELM3002_B416BFEF;
	{attribute addProperty Name "A_0002(ELM3002-0000-0017)"}
	{attribute addProperty PreviousPort "A_0001(ELM3002-0000-0016) : B"}
	A_0002_ELM3002_0000_0017 : ELM3002_B416BFEF;
	{attribute addProperty Name "A_0003(ELM3002-0000-0018)"}
	{attribute addProperty PreviousPort "A_0002(ELM3002-0000-0017) : B"}
	A_0003_ELM3002_0000_0018 : ELM3002_B416BFEF;
	{attribute addProperty Name "A_0004(ELM3004-0000-0016)"}
	{attribute addProperty PreviousPort "A_0003(ELM3002-0000-0018) : B"}
	A_0004_ELM3004_0000_0016 : ELM3004_9E251EA4;
	{attribute addProperty Name "A_0005(ELM3004-0000-0017)"}
	{attribute addProperty PreviousPort "A_0004(ELM3004-0000-0016) : B"}
	A_0005_ELM3004_0000_0017 : ELM3004_9E251EA4;
	{attribute addProperty Name "A_0006(ELM3004-0000-0018)"}
	{attribute addProperty PreviousPort "A_0005(ELM3004-0000-0017) : B"}
	A_0006_ELM3004_0000_0018 : ELM3004_9E251EA4;
	{attribute addProperty Name "A_0007(ELM3004-0000-0019)"}
	{attribute addProperty PreviousPort "A_0006(ELM3004-0000-0018) : B"}
	A_0007_ELM3004_0000_0019 : ELM3004_9E251EA4;
END_STRUCT
END_TYPE

// ---- DUTs/IO/Topology/Beckhoff_ELM31xxEK1122_DD495580.TcDUT
{attribute 'GeneratedUsingTerminal: EK1122-0000-0018'}
{attribute addProperty BoxType "EK1122-0000-0018"}
{attribute addProperty Id "Beckhoff_ELM31xxsub_EK1100EK1100_1FC0878B2"}
{attribute addProperty CRC "3712570752"}
{attribute addProperty Size "2"}
{attribute addProperty Name "Beckhoff ELM31xxEK1122"}
TYPE Beckhoff_ELM31xxEK1122_DD495580 EXTENDS EK1122_1FC0878B :
STRUCT
	{attribute addProperty Name "Beckhoff ELM31xxsub EK1100"}
	{attribute addProperty PreviousPort "Beckhoff ELM31xxEK1122 : D"}
	Beckhoff_ELM31xxsub_EK1100 : EK1100_1FC0878B;
END_STRUCT
END_TYPE

// ---- DUTs/IO/Topology/Beckhoff_ELM31xx_96F66E1E.TcDUT
{attribute 'GeneratedUsingTerminal: EK1100-0000-0018'}
{attribute addProperty BoxType "EK1100-0000-0018"}
{attribute addProperty Id "Beckhoff_ELM31xxEK1122Beckhoff_ELM31xxEK1122_DD4955802A_0001_ELM3102_0000_0016ELM3102_B416BFEF50A_0002_ELM3102_0000_0017ELM3102_B416BFEF50A_0003_ELM3102_0000_0018ELM3102_B416BFEF50A_0004_ELM3104_0000_0016ELM3104_9E251EA472A_0005_ELM3104_0000_0017ELM3104_9E251EA472A_0006_ELM3104_0000_0018ELM3104_9E251EA472A_0007_ELM3142_0000_0016ELM3142_B416BFEF50A_0008_ELM3142_0000_0017ELM3142_B416BFEF50A_0009_ELM3144_0000_0016ELM3144_9E251EA472A_0010_ELM3144_0000_0017ELM3144_9E251EA472A_0011_ELM3146_0000_0016ELM3146_EA6DB5D794A_0012_ELM3146_0000_0017ELM3146_EA6DB5D794A_0013_ELM3146_0000_0018ELM3146_EA6DB5D794A_0014_ELM3148_0000_0017ELM3148_0838C628116A_0015_ELM3148_0000_0018ELM3148_0838C628116A_0016_ELM3148_0000_0019ELM3148_0838C628116"}
{attribute addProperty CRC "2532732446"}
{attribute addProperty Size "1242"}
{attribute addProperty Name "Beckhoff ELM31xx"}
TYPE Beckhoff_ELM31xx_96F66E1E EXTENDS EK1100_1FC0878B :
STRUCT
	{attribute addProperty Name "Beckhoff ELM31xxEK1122"}
	{attribute addProperty PreviousPort "Beckhoff ELM31xx : B"}
	Beckhoff_ELM31xxEK1122 : Beckhoff_ELM31xxEK1122_DD495580;
	{attribute addProperty Name "A_0001(ELM3102-0000-0016)"}
	{attribute addProperty PreviousPort "Beckhoff ELM31xxEK1122 : C"}
	A_0001_ELM3102_0000_0016 : ELM3102_B416BFEF;
	{attribute addProperty Name "A_0002(ELM3102-0000-0017)"}
	{attribute addProperty PreviousPort "A_0001(ELM3102-0000-0016) : B"}
	A_0002_ELM3102_0000_0017 : ELM3102_B416BFEF;
	{attribute addProperty Name "A_0003(ELM3102-0000-0018)"}
	{attribute addProperty PreviousPort "A_0002(ELM3102-0000-0017) : B"}
	A_0003_ELM3102_0000_0018 : ELM3102_B416BFEF;
	{attribute addProperty Name "A_0004(ELM3104-0000-0016)"}
	{attribute addProperty PreviousPort "A_0003(ELM3102-0000-0018) : B"}
	A_0004_ELM3104_0000_0016 : ELM3104_9E251EA4;
	{attribute addProperty Name "A_0005(ELM3104-0000-0017)"}
	{attribute addProperty PreviousPort "A_0004(ELM3104-0000-0016) : B"}
	A_0005_ELM3104_0000_0017 : ELM3104_9E251EA4;
	{attribute addProperty Name "A_0006(ELM3104-0000-0018)"}
	{attribute addProperty PreviousPort "A_0005(ELM3104-0000-0017) : B"}
	A_0006_ELM3104_0000_0018 : ELM3104_9E251EA4;
	{attribute addProperty Name "A_0007(ELM3142-0000-0016)"}
	{attribute addProperty PreviousPort "A_0006(ELM3104-0000-0018) : B"}
	A_0007_ELM3142_0000_0016 : ELM3142_B416BFEF;
	{attribute addProperty Name "A_0008(ELM3142-0000-0017)"}
	{attribute addProperty PreviousPort "A_0007(ELM3142-0000-0016) : B"}
	A_0008_ELM3142_0000_0017 : ELM3142_B416BFEF;
	{attribute addProperty Name "A_0009(ELM3144-0000-0016)"}
	{attribute addProperty PreviousPort "A_0008(ELM3142-0000-0017) : B"}
	A_0009_ELM3144_0000_0016 : ELM3144_9E251EA4;
	{attribute addProperty Name "A_0010(ELM3144-0000-0017)"}
	{attribute addProperty PreviousPort "A_0009(ELM3144-0000-0016) : B"}
	A_0010_ELM3144_0000_0017 : ELM3144_9E251EA4;
	{attribute addProperty Name "A_0011(ELM3146-0000-0016)"}
	{attribute addProperty PreviousPort "A_0010(ELM3144-0000-0017) : B"}
	A_0011_ELM3146_0000_0016 : ELM3146_EA6DB5D7;
	{attribute addProperty Name "A_0012(ELM3146-0000-0017)"}
	{attribute addProperty PreviousPort "A_0011(ELM3146-0000-0016) : B"}
	A_0012_ELM3146_0000_0017 : ELM3146_EA6DB5D7;
	{attribute addProperty Name "A_0013(ELM3146-0000-0018)"}
	{attribute addProperty PreviousPort "A_0012(ELM3146-0000-0017) : B"}
	A_0013_ELM3146_0000_0018 : ELM3146_EA6DB5D7;
	{attribute addProperty Name "A_0014(ELM3148-0000-0017)"}
	{attribute addProperty PreviousPort "A_0013(ELM3146-0000-0018) : B"}
	A_0014_ELM3148_0000_0017 : ELM3148_0838C628;
	{attribute addProperty Name "A_0015(ELM3148-0000-0018)"}
	{attribute addProperty PreviousPort "A_0014(ELM3148-0000-0017) : B"}
	A_0015_ELM3148_0000_0018 : ELM3148_0838C628;
	{attribute addProperty Name "A_0016(ELM3148-0000-0019)"}
	{attribute addProperty PreviousPort "A_0015(ELM3148-0000-0018) : B"}
	A_0016_ELM3148_0000_0019 : ELM3148_0838C628;
END_STRUCT
END_TYPE

// ---- DUTs/IO/Topology/Beckhoff_ELM35xxEK1122_0F7152EB.TcDUT
{attribute 'GeneratedUsingTerminal: EK1122-0000-0018'}
{attribute addProperty BoxType "EK1122-0000-0018"}
{attribute addProperty Id "Beckhoff_ELM35xxsub_EK1100EK1100_1FC0878B2"}
{attribute addProperty CRC "259085035"}
{attribute addProperty Size "2"}
{attribute addProperty Name "Beckhoff ELM35xxEK1122"}
TYPE Beckhoff_ELM35xxEK1122_0F7152EB EXTENDS EK1122_1FC0878B :
STRUCT
	{attribute addProperty Name "Beckhoff ELM35xxsub EK1100"}
	{attribute addProperty PreviousPort "Beckhoff ELM35xxEK1122 : D"}
	Beckhoff_ELM35xxsub_EK1100 : EK1100_1FC0878B;
END_STRUCT
END_TYPE

// ---- DUTs/IO/Topology/Beckhoff_ELM35xx_B8844D22.TcDUT
{attribute 'GeneratedUsingTerminal: EK1100-0000-0018'}
{attribute addProperty BoxType "EK1100-0000-0018"}
{attribute addProperty Id "Beckhoff_ELM35xxEK1122Beckhoff_ELM35xxEK1122_0F7152EB2A_0001_ELM3502_0000_0016ELM3502_B416BFEF50A_0002_ELM3502_0000_0017ELM3502_B416BFEF50A_0003_ELM3502_0000_0018ELM3502_B416BFEF50A_0004_ELM3502_0000_0019ELM3502_B416BFEF50A_0005_ELM3504_0000_0016ELM3504_9E251EA472A_0006_ELM3504_0000_0017ELM3504_9E251EA472A_0007_ELM3504_0000_0018ELM3504_9E251EA472A_0008_ELM3504_0000_0019ELM3504_9E251EA472"}
{attribute addProperty CRC "3095678242"}
{attribute addProperty Size "490"}
{attribute addProperty Name "Beckhoff ELM35xx"}
TYPE Beckhoff_ELM35xx_B8844D22 EXTENDS EK1100_1FC0878B :
STRUCT
	{attribute addProperty Name "Beckhoff ELM35xxEK1122"}
	{attribute addProperty PreviousPort "Beckhoff ELM35xx : B"}
	Beckhoff_ELM35xxEK1122 : Beckhoff_ELM35xxEK1122_0F7152EB;
	{attribute addProperty Name "A_0001(ELM3502-0000-0016)"}
	{attribute addProperty PreviousPort "Beckhoff ELM35xxEK1122 : C"}
	A_0001_ELM3502_0000_0016 : ELM3502_B416BFEF;
	{attribute addProperty Name "A_0002(ELM3502-0000-0017)"}
	{attribute addProperty PreviousPort "A_0001(ELM3502-0000-0016) : B"}
	A_0002_ELM3502_0000_0017 : ELM3502_B416BFEF;
	{attribute addProperty Name "A_0003(ELM3502-0000-0018)"}
	{attribute addProperty PreviousPort "A_0002(ELM3502-0000-0017) : B"}
	A_0003_ELM3502_0000_0018 : ELM3502_B416BFEF;
	{attribute addProperty Name "A_0004(ELM3502-0000-0019)"}
	{attribute addProperty PreviousPort "A_0003(ELM3502-0000-0018) : B"}
	A_0004_ELM3502_0000_0019 : ELM3502_B416BFEF;
	{attribute addProperty Name "A_0005(ELM3504-0000-0016)"}
	{attribute addProperty PreviousPort "A_0004(ELM3502-0000-0019) : B"}
	A_0005_ELM3504_0000_0016 : ELM3504_9E251EA4;
	{attribute addProperty Name "A_0006(ELM3504-0000-0017)"}
	{attribute addProperty PreviousPort "A_0005(ELM3504-0000-0016) : B"}
	A_0006_ELM3504_0000_0017 : ELM3504_9E251EA4;
	{attribute addProperty Name "A_0007(ELM3504-0000-0018)"}
	{attribute addProperty PreviousPort "A_0006(ELM3504-0000-0017) : B"}
	A_0007_ELM3504_0000_0018 : ELM3504_9E251EA4;
	{attribute addProperty Name "A_0008(ELM3504-0000-0019)"}
	{attribute addProperty PreviousPort "A_0007(ELM3504-0000-0018) : B"}
	A_0008_ELM3504_0000_0019 : ELM3504_9E251EA4;
END_STRUCT
END_TYPE

// ---- DUTs/IO/Topology/Beckhoff_ELM36xxEK1122_91B39932.TcDUT
{attribute 'GeneratedUsingTerminal: EK1122-0000-0018'}
{attribute addProperty BoxType "EK1122-0000-0018"}
{attribute addProperty Id "Beckhoff_ELM36xxsub_EK1100EK1100_1FC0878B2"}
{attribute addProperty CRC "2444466482"}
{attribute addProperty Size "2"}
{attribute addProperty Name "Beckhoff ELM36xxEK1122"}
TYPE Beckhoff_ELM36xxEK1122_91B39932 EXTENDS EK1122_1FC0878B :
STRUCT
	{attribute addProperty Name "Beckhoff ELM36xxsub EK1100"}
	{attribute addProperty PreviousPort "Beckhoff ELM36xxEK1122 : D"}
	Beckhoff_ELM36xxsub_EK1100 : EK1100_1FC0878B;
END_STRUCT
END_TYPE

// ---- DUTs/IO/Topology/Beckhoff_ELM36xx_2C7C6FAB.TcDUT
{attribute 'GeneratedUsingTerminal: EK1100-0000-0018'}
{attribute addProperty BoxType "EK1100-0000-0018"}
{attribute addProperty Id "Beckhoff_ELM36xxEK1122Beckhoff_ELM36xxEK1122_91B399322A_0001_ELM3602_0000_0017ELM3602_B416BFEF50A_0002_ELM3602_0000_0018ELM3602_B416BFEF50A_0003_ELM3602_0002_0016ELM3602_B416BFEF50A_0004_ELM3602_0002_0017ELM3602_B416BFEF50A_0005_ELM3602_0002_0018ELM3602_B416BFEF50A_0006_ELM3604_0000_0017ELM3604_9E251EA472A_0007_ELM3604_0000_0018ELM3604_9E251EA472A_0008_ELM3604_0002_0016ELM3604_9E251EA472A_0009_ELM3604_0002_0017ELM3604_9E251EA472A_0010_ELM3604_0002_0018ELM3604_9E251EA472"}
{attribute addProperty CRC "746352555"}
{attribute addProperty Size "612"}
{attribute addProperty Name "Beckhoff ELM36xx"}
TYPE Beckhoff_ELM36xx_2C7C6FAB EXTENDS EK1100_1FC0878B :
STRUCT
	{attribute addProperty Name "Beckhoff ELM36xxEK1122"}
	{attribute addProperty PreviousPort "Beckhoff ELM36xx : B"}
	Beckhoff_ELM36xxEK1122 : Beckhoff_ELM36xxEK1122_91B39932;
	{attribute addProperty Name "A_0001(ELM3602-0000-0017)"}
	{attribute addProperty PreviousPort "Beckhoff ELM36xxEK1122 : C"}
	A_0001_ELM3602_0000_0017 : ELM3602_B416BFEF;
	{attribute addProperty Name "A_0002(ELM3602-0000-0018)"}
	{attribute addProperty PreviousPort "A_0001(ELM3602-0000-0017) : B"}
	A_0002_ELM3602_0000_0018 : ELM3602_B416BFEF;
	{attribute addProperty Name "A_0003(ELM3602-0002-0016)"}
	{attribute addProperty PreviousPort "A_0002(ELM3602-0000-0018) : B"}
	A_0003_ELM3602_0002_0016 : ELM3602_B416BFEF;
	{attribute addProperty Name "A_0004(ELM3602-0002-0017)"}
	{attribute addProperty PreviousPort "A_0003(ELM3602-0002-0016) : B"}
	A_0004_ELM3602_0002_0017 : ELM3602_B416BFEF;
	{attribute addProperty Name "A_0005(ELM3602-0002-0018)"}
	{attribute addProperty PreviousPort "A_0004(ELM3602-0002-0017) : B"}
	A_0005_ELM3602_0002_0018 : ELM3602_B416BFEF;
	{attribute addProperty Name "A_0006(ELM3604-0000-0017)"}
	{attribute addProperty PreviousPort "A_0005(ELM3602-0002-0018) : B"}
	A_0006_ELM3604_0000_0017 : ELM3604_9E251EA4;
	{attribute addProperty Name "A_0007(ELM3604-0000-0018)"}
	{attribute addProperty PreviousPort "A_0006(ELM3604-0000-0017) : B"}
	A_0007_ELM3604_0000_0018 : ELM3604_9E251EA4;
	{attribute addProperty Name "A_0008(ELM3604-0002-0016)"}
	{attribute addProperty PreviousPort "A_0007(ELM3604-0000-0018) : B"}
	A_0008_ELM3604_0002_0016 : ELM3604_9E251EA4;
	{attribute addProperty Name "A_0009(ELM3604-0002-0017)"}
	{attribute addProperty PreviousPort "A_0008(ELM3604-0002-0016) : B"}
	A_0009_ELM3604_0002_0017 : ELM3604_9E251EA4;
	{attribute addProperty Name "A_0010(ELM3604-0002-0018)"}
	{attribute addProperty PreviousPort "A_0009(ELM3604-0002-0017) : B"}
	A_0010_ELM3604_0002_0018 : ELM3604_9E251EA4;
END_STRUCT
END_TYPE

// ---- DUTs/IO/Topology/Beckhoff_ELM37xxEK1122_E40DDF85.TcDUT
{attribute 'GeneratedUsingTerminal: EK1122-0000-0018'}
{attribute addProperty BoxType "EK1122-0000-0018"}
{attribute addProperty Id "Beckhoff_ELM37xxsub_EK1100EK1100_1FC0878B2"}
{attribute addProperty CRC "3826114437"}
{attribute addProperty Size "2"}
{attribute addProperty Name "Beckhoff ELM37xxEK1122"}
TYPE Beckhoff_ELM37xxEK1122_E40DDF85 EXTENDS EK1122_1FC0878B :
STRUCT
	{attribute addProperty Name "Beckhoff ELM37xxsub EK1100"}
	{attribute addProperty PreviousPort "Beckhoff ELM37xxEK1122 : D"}
	Beckhoff_ELM37xxsub_EK1100 : EK1100_1FC0878B;
END_STRUCT
END_TYPE

// ---- DUTs/IO/Topology/Beckhoff_ELM37xx_73C6C048.TcDUT
{attribute 'GeneratedUsingTerminal: EK1100-0000-0018'}
{attribute addProperty BoxType "EK1100-0000-0018"}
{attribute addProperty Id "Beckhoff_ELM37xxEK1122Beckhoff_ELM37xxEK1122_E40DDF852A_0001_ELM3702_0000_0016ELM3702_B416BFEF50A_0002_ELM3702_0000_0017ELM3702_B416BFEF50A_0003_ELM3704_0000_0016ELM3704_9E251EA472A_0004_ELM3704_0000_0017ELM3704_9E251EA472A_0005_ELM3704_0001_0017ELM3704_9E251EA472A_0006_ELM3704_0020_0016ELM3704_9E251EA472A_0007_ELM3702_0101_0016ELM3702_B416BFEF50A_0008_ELM3704_1001_0016ELM3704_9E251EA472A_0009_ELM3704_1001_0017ELM3704_9E251EA472"}
{attribute addProperty CRC "1942405192"}
{attribute addProperty Size "584"}
{attribute addProperty Name "Beckhoff ELM37xx"}
TYPE Beckhoff_ELM37xx_73C6C048 EXTENDS EK1100_1FC0878B :
STRUCT
	{attribute addProperty Name "Beckhoff ELM37xxEK1122"}
	{attribute addProperty PreviousPort "Beckhoff ELM37xx : B"}
	Beckhoff_ELM37xxEK1122 : Beckhoff_ELM37xxEK1122_E40DDF85;
	{attribute addProperty Name "A_0001(ELM3702-0000-0016)"}
	{attribute addProperty PreviousPort "Beckhoff ELM37xxEK1122 : C"}
	A_0001_ELM3702_0000_0016 : ELM3702_B416BFEF;
	{attribute addProperty Name "A_0002(ELM3702-0000-0017)"}
	{attribute addProperty PreviousPort "A_0001(ELM3702-0000-0016) : B"}
	A_0002_ELM3702_0000_0017 : ELM3702_B416BFEF;
	{attribute addProperty Name "A_0003(ELM3704-0000-0016)"}
	{attribute addProperty PreviousPort "A_0002(ELM3702-0000-0017) : B"}
	A_0003_ELM3704_0000_0016 : ELM3704_9E251EA4;
	{attribute addProperty Name "A_0004(ELM3704-0000-0017)"}
	{attribute addProperty PreviousPort "A_0003(ELM3704-0000-0016) : B"}
	A_0004_ELM3704_0000_0017 : ELM3704_9E251EA4;
	{attribute addProperty Name "A_0005(ELM3704-0001-0017)"}
	{attribute addProperty PreviousPort "A_0004(ELM3704-0000-0017) : B"}
	A_0005_ELM3704_0001_0017 : ELM3704_9E251EA4;
	{attribute addProperty Name "A_0006(ELM3704-0020-0016)"}
	{attribute addProperty PreviousPort "A_0005(ELM3704-0001-0017) : B"}
	A_0006_ELM3704_0020_0016 : ELM3704_9E251EA4;
	{attribute addProperty Name "A_0007(ELM3702-0101-0016)"}
	{attribute addProperty PreviousPort "A_0006(ELM3704-0020-0016) : B"}
	A_0007_ELM3702_0101_0016 : ELM3702_B416BFEF;
	{attribute addProperty Name "A_0008(ELM3704-1001-0016)"}
	{attribute addProperty PreviousPort "A_0007(ELM3702-0101-0016) : B"}
	A_0008_ELM3704_1001_0016 : ELM3704_9E251EA4;
	{attribute addProperty Name "A_0009(ELM3704-1001-0017)"}
	{attribute addProperty PreviousPort "A_0008(ELM3704-1001-0016) : B"}
	A_0009_ELM3704_1001_0017 : ELM3704_9E251EA4;
END_STRUCT
END_TYPE

// ---- DUTs/IO/Topology/Beckhoff_ELM3xxx_0030EK1122_95B17030.TcDUT
{attribute 'GeneratedUsingTerminal: EK1122-0000-0018'}
{attribute addProperty BoxType "EK1122-0000-0018"}
{attribute addProperty Id "Beckhoff_ELM3xxx_0030sub_EK1100EK1100_1FC0878B2"}
{attribute addProperty CRC "2511433776"}
{attribute addProperty Size "2"}
{attribute addProperty Name "Beckhoff ELM3xxx-0030EK1122"}
TYPE Beckhoff_ELM3xxx_0030EK1122_95B17030 EXTENDS EK1122_1FC0878B :
STRUCT
	{attribute addProperty Name "Beckhoff ELM3xxx-0030sub EK1100"}
	{attribute addProperty PreviousPort "Beckhoff ELM3xxx-0030EK1122 : D"}
	Beckhoff_ELM3xxx_0030sub_EK1100 : EK1100_1FC0878B;
END_STRUCT
END_TYPE

// ---- DUTs/IO/Topology/Beckhoff_ELM3xxx_0030_615BF1E1.TcDUT
{attribute 'GeneratedUsingTerminal: EK1100-0000-0018'}
{attribute addProperty BoxType "EK1100-0000-0018"}
{attribute addProperty Id "Beckhoff_ELM3xxx_0030EK1122Beckhoff_ELM3xxx_0030EK1122_95B170302A_0001_ELM3002_0030_0017ELM3002_B416BFEF50A_0002_ELM3002_0030_0018ELM3002_B416BFEF50A_0003_ELM3004_0030_0018ELM3004_9E251EA472A_0004_ELM3004_0030_0019ELM3004_9E251EA472A_0005_ELM3502_0030_0019ELM3502_B416BFEF50A_0006_ELM3504_0030_0019ELM3504_9E251EA472"}
{attribute addProperty CRC "1633415649"}
{attribute addProperty Size "368"}
{attribute addProperty Name "Beckhoff ELM3xxx-0030"}
TYPE Beckhoff_ELM3xxx_0030_615BF1E1 EXTENDS EK1100_1FC0878B :
STRUCT
	{attribute addProperty Name "Beckhoff ELM3xxx-0030EK1122"}
	{attribute addProperty PreviousPort "Beckhoff ELM3xxx-0030 : B"}
	Beckhoff_ELM3xxx_0030EK1122 : Beckhoff_ELM3xxx_0030EK1122_95B17030;
	{attribute addProperty Name "A_0001(ELM3002-0030-0017)"}
	{attribute addProperty PreviousPort "Beckhoff ELM3xxx-0030EK1122 : C"}
	A_0001_ELM3002_0030_0017 : ELM3002_B416BFEF;
	{attribute addProperty Name "A_0002(ELM3002-0030-0018)"}
	{attribute addProperty PreviousPort "A_0001(ELM3002-0030-0017) : B"}
	A_0002_ELM3002_0030_0018 : ELM3002_B416BFEF;
	{attribute addProperty Name "A_0003(ELM3004-0030-0018)"}
	{attribute addProperty PreviousPort "A_0002(ELM3002-0030-0018) : B"}
	A_0003_ELM3004_0030_0018 : ELM3004_9E251EA4;
	{attribute addProperty Name "A_0004(ELM3004-0030-0019)"}
	{attribute addProperty PreviousPort "A_0003(ELM3004-0030-0018) : B"}
	A_0004_ELM3004_0030_0019 : ELM3004_9E251EA4;
	{attribute addProperty Name "A_0005(ELM3502-0030-0019)"}
	{attribute addProperty PreviousPort "A_0004(ELM3004-0030-0019) : B"}
	A_0005_ELM3502_0030_0019 : ELM3502_B416BFEF;
	{attribute addProperty Name "A_0006(ELM3504-0030-0019)"}
	{attribute addProperty PreviousPort "A_0005(ELM3502-0030-0019) : B"}
	A_0006_ELM3504_0030_0019 : ELM3504_9E251EA4;
END_STRUCT
END_TYPE

// ---- DUTs/IO/Topology/Beckhoff_ELM9xxxEK1122_C8584423.TcDUT
{attribute 'GeneratedUsingTerminal: EK1122-0000-0018'}
{attribute addProperty BoxType "EK1122-0000-0018"}
{attribute addProperty Id "Beckhoff_ELM9xxxsub_EK1100EK1100_1FC0878B2"}
{attribute addProperty CRC "3361227811"}
{attribute addProperty Size "2"}
{attribute addProperty Name "Beckhoff ELM9xxxEK1122"}
TYPE Beckhoff_ELM9xxxEK1122_C8584423 EXTENDS EK1122_1FC0878B :
STRUCT
	{attribute addProperty Name "Beckhoff ELM9xxxsub EK1100"}
	{attribute addProperty PreviousPort "Beckhoff ELM9xxxEK1122 : D"}
	Beckhoff_ELM9xxxsub_EK1100 : EK1100_1FC0878B;
END_STRUCT
END_TYPE

// ---- DUTs/IO/Topology/Beckhoff_ELM9xxx_3A75798B.TcDUT
{attribute 'GeneratedUsingTerminal: EK1100-0000-0018'}
{attribute addProperty BoxType "EK1100-0000-0018"}
{attribute addProperty Id "Beckhoff_ELM9xxxEK1122Beckhoff_ELM9xxxEK1122_C85844232A_0002_ELM9410_0000_0016ELM9410_DD55393581A_0003_ELM9410_0000_0017ELM9410_DD55393581A_0004_ELM9410_0000_0018ELM9410_DD55393581A_0005_ELM9410_0000_0019ELM9410_DD55393581A_0006_ELM9410_0000_0020ELM9410_DD55393581"}
{attribute addProperty CRC "980777355"}
{attribute addProperty Size "407"}
{attribute addProperty Name "Beckhoff ELM9xxx"}
TYPE Beckhoff_ELM9xxx_3A75798B EXTENDS EK1100_1FC0878B :
STRUCT
	{attribute addProperty Name "Beckhoff ELM9xxxEK1122"}
	{attribute addProperty PreviousPort "Beckhoff ELM9xxx : B"}
	Beckhoff_ELM9xxxEK1122 : Beckhoff_ELM9xxxEK1122_C8584423;
	{attribute addProperty Name "A_0002(ELM9410-0000-0016)"}
	{attribute addProperty PreviousPort "Beckhoff ELM9xxxEK1122 : C"}
	A_0002_ELM9410_0000_0016 : ELM9410_DD553935;
	{attribute addProperty Name "A_0003(ELM9410-0000-0017)"}
	{attribute addProperty PreviousPort "A_0002(ELM9410-0000-0016) : B"}
	A_0003_ELM9410_0000_0017 : ELM9410_DD553935;
	{attribute addProperty Name "A_0004(ELM9410-0000-0018)"}
	{attribute addProperty PreviousPort "A_0003(ELM9410-0000-0017) : B"}
	A_0004_ELM9410_0000_0018 : ELM9410_DD553935;
	{attribute addProperty Name "A_0005(ELM9410-0000-0019)"}
	{attribute addProperty PreviousPort "A_0004(ELM9410-0000-0018) : B"}
	A_0005_ELM9410_0000_0019 : ELM9410_DD553935;
	{attribute addProperty Name "A_0006(ELM9410-0000-0020)"}
	{attribute addProperty PreviousPort "A_0005(ELM9410-0000-0019) : B"}
	A_0006_ELM9410_0000_0020 : ELM9410_DD553935;
END_STRUCT
END_TYPE

// ---- DUTs/IO/Topology/EtherCAT_Master_ELMxxxx_56F7A9AD.TcDUT
{attribute 'GeneratedUsingTerminal: IODEVICETYPE_ETHERCATPROT'}
{attribute addProperty BoxType "IODEVICETYPE_ETHERCATPROT"}
{attribute addProperty Id "Beckhoff_ELM3xxxBeckhoff_ELM3xxx_31A44528440Beckhoff_ELM31xxBeckhoff_ELM31xx_96F66E1E1242Beckhoff_ELM35xxBeckhoff_ELM35xx_B8844D22490Beckhoff_ELM36xxBeckhoff_ELM36xx_2C7C6FAB612Beckhoff_ELM37xxBeckhoff_ELM37xx_73C6C048584Beckhoff_ELM3xxx_0030Beckhoff_ELM3xxx_0030_615BF1E1368Beckhoff_ELM9xxxBeckhoff_ELM9xxx_3A75798B407SyncUnitsSyncUnits_99E584AF18InputsInputs_25A0042B160OutputsOutputs_2397A10E106InfoDataInfoData_E68C61CD28"}
{attribute addProperty CRC "1459071405"}
{attribute addProperty Size "4455"}
{attribute addProperty Name "EtherCAT Master ELMxxxx"}
TYPE EtherCAT_Master_ELMxxxx_56F7A9AD EXTENDS EtcMasterBase_62654B43 :
STRUCT
	{attribute addProperty Name "Beckhoff ELM3xxx"}
	{attribute addProperty PreviousPort "EtherCAT Master ELMxxxx : Master"}
	Beckhoff_ELM3xxx : Beckhoff_ELM3xxx_31A44528;
	{attribute addProperty Name "Beckhoff ELM31xx"}
	{attribute addProperty PreviousPort "Beckhoff ELM3xxx : C"}
	Beckhoff_ELM31xx : Beckhoff_ELM31xx_96F66E1E;
	{attribute addProperty Name "Beckhoff ELM35xx"}
	{attribute addProperty PreviousPort "Beckhoff ELM31xx : C"}
	Beckhoff_ELM35xx : Beckhoff_ELM35xx_B8844D22;
	{attribute addProperty Name "Beckhoff ELM36xx"}
	{attribute addProperty PreviousPort "Beckhoff ELM35xx : C"}
	Beckhoff_ELM36xx : Beckhoff_ELM36xx_2C7C6FAB;
	{attribute addProperty Name "Beckhoff ELM37xx"}
	{attribute addProperty PreviousPort "Beckhoff ELM36xx : C"}
	Beckhoff_ELM37xx : Beckhoff_ELM37xx_73C6C048;
	{attribute addProperty Name "Beckhoff ELM3xxx-0030"}
	{attribute addProperty PreviousPort "Beckhoff ELM37xx : C"}
	Beckhoff_ELM3xxx_0030 : Beckhoff_ELM3xxx_0030_615BF1E1;
	{attribute addProperty Name "Beckhoff ELM9xxx"}
	{attribute addProperty PreviousPort "Beckhoff ELM3xxx-0030 : C"}
	Beckhoff_ELM9xxx : Beckhoff_ELM9xxx_3A75798B;
	{attribute addProperty Name "SyncUnits"}
	SyncUnits : SyncUnits_99E584AF;
	{attribute addProperty Name "Inputs"}
	Inputs : Inputs_25A0042B;
	{attribute addProperty Name "Outputs"}
	Outputs : Outputs_2397A10E;
	{attribute addProperty Name "InfoData"}
	InfoData : InfoData_E68C61CD;
END_STRUCT
END_TYPE

// ---- DUTs/IO/Base/EtcSlaveBase_82538BE2.TcDUT

TYPE EtcSlaveBase_82538BE2 :
STRUCT
END_STRUCT
END_TYPE

// ---- DUTs/IO/Base/EtcSlaveBase_82538BE2.TcDUT

TYPE EtcSlaveBase_82538BE2 :
STRUCT
END_STRUCT
END_TYPE

// ---- DUTs/IO/Base/EtcSlaveBase_82538BE2.TcDUT

TYPE EtcSlaveBase_82538BE2 :
STRUCT
END_STRUCT
END_TYPE

// ---- DUTs/IO/Base/EtcSlaveTerminalBase_947E5A46.TcDUT

{attribute clr[Container(Layout.Stack)]}
{attribute clr[Group(Layout.GroupBox)]}
{attribute addProperty PreviousPort "Unknown"}
TYPE EtcSlaveTerminalBase_947E5A46 EXTENDS EtcSlaveBase_82538BE2 :
STRUCT
END_STRUCT
END_TYPE

// ---- DUTs/IO/Base/EtcSlaveBoxBase_77A0E4A7.TcDUT

{attribute clr[Container(Layout.Stack)]}
{attribute clr[Group(Layout.GroupBox)]}
{attribute addProperty PreviousPort "Unknown"}
TYPE EtcSlaveBoxBase_77A0E4A7 EXTENDS EtcSlaveBase_82538BE2 :
STRUCT
END_STRUCT
END_TYPE

// ---- DUTs/IO/Base/EtcSlaveEndTerminalBase_866C7F0C.TcDUT

{attribute clr[Container(Layout.Stack)]}
{attribute clr[Group(Layout.GroupBox)]}
{attribute addProperty PreviousPort "Unknown"}
TYPE EtcSlaveEndTerminalBase_866C7F0C EXTENDS EtcSlaveBase_82538BE2 :
STRUCT
END_STRUCT
END_TYPE

// ---- DUTs/IO/Base/InputBase_8311D824.TcDUT

TYPE InputBase_8311D824 :
STRUCT
END_STRUCT
END_TYPE

// ---- DUTs/IO/Base/OutputBase_10CEE7DE.TcDUT

TYPE OutputBase_10CEE7DE :
STRUCT
END_STRUCT
END_TYPE

// ---- DUTs/IO/Base/EtcMasterBase_62654B43.TcDUT

TYPE EtcMasterBase_62654B43 :
STRUCT
END_STRUCT
END_TYPE

// ---- GVLs/GVL_iXlinker.TcGVL
{attribute 'qualified_only'}
VAR_GLOBAL
		EtherCAT_Master_ELMxxxx : EtherCAT_Master_ELMxxxx_56F7A9AD;
END_VAR

// ---- POUs/MAIN.TcPOU
PROGRAM MAIN
VAR
END_VAR

END_PROGRAM
